LIN {X 0,Y 584.039,Z 358.291,A -85,B 0,C 180,E1 26452.128,E2 26452.128} C_VEL
LIN {X 0,Y 584.089,Z 358.294,A -85,B 0,C 180,E1 26449.046,E2 26449.046} C_VEL
LIN {X 0,Y 584.1,Z 358.289,A -85,B 0,C 180,E1 26446.664,E2 26446.664} C_VEL
LIN {X 0,Y 583.093,Z 358.412,A -85,B 0,C 180,E1 26445.909,E2 26445.909} C_VEL
LIN {X 0,Y 576.621,Z 359.216,A -85,B 0,C 180,E1 26443.789,E2 26443.789} C_VEL
LIN {X 0,Y 576.118,Z 359.28,A -85,B 0,C 180,E1 26443.236,E2 26443.236} C_VEL
LIN {X 0,Y 576.115,Z 359.276,A -85,B 0,C 180,E1 26439.857,E2 26439.857} C_VEL
LIN {X 0,Y 576.157,Z 359.281,A -85,B 0,C 180,E1 26436.692,E2 26436.692} C_VEL
LIN {X 0,Y 576.112,Z 359.278,A -85,B 0,C 180,E1 26433.51,E2 26433.51} C_VEL
LIN {X 0,Y 576.159,Z 359.278,A -85,B 0,C 180,E1 26430.357,E2 26430.357} C_VEL
LIN {X 0,Y 576.115,Z 359.28,A -85,B 0,C 180,E1 26427.131,E2 26427.131} C_VEL
LIN {X 0,Y 576.159,Z 359.276,A -85,B 0,C 180,E1 26423.961,E2 26423.961} C_VEL
LIN {X 0,Y 576.126,Z 359.281,A -85,B 0,C 180,E1 26420.71,E2 26420.71} C_VEL
LIN {X 0,Y 576.141,Z 359.275,A -85,B 0,C 180,E1 26417.371,E2 26417.371} C_VEL
LIN {X 0,Y 576.158,Z 359.281,A -85,B 0,C 180,E1 26414.073,E2 26414.073} C_VEL
LIN {X 0,Y 576.126,Z 359.278,A -85,B 0,C 180,E1 26410.828,E2 26410.828} C_VEL
LIN {X 0,Y 576.153,Z 359.277,A -85,B 0,C 180,E1 26407.647,E2 26407.647} C_VEL
LIN {X 0,Y 576.129,Z 359.278,A -85,B 0,C 180,E1 26404.451,E2 26404.451} C_VEL
LIN {X 0,Y 576.155,Z 359.268,A -85,B 0,C 180,E1 26401.179,E2 26401.179} C_VEL
LIN {X 0,Y 576.151,Z 359.283,A -85,B 0,C 180,E1 26397.824,E2 26397.824} C_VEL
LIN {X 0,Y 576.139,Z 359.274,A -85,B 0,C 180,E1 26394.501,E2 26394.501} C_VEL
LIN {X 0,Y 576.147,Z 359.275,A -85,B 0,C 180,E1 26391.263,E2 26391.263} C_VEL
LIN {X 0,Y 576.137,Z 359.279,A -85,B 0,C 180,E1 26388.005,E2 26388.005} C_VEL
LIN {X 0,Y 576.147,Z 359.274,A -85,B 0,C 180,E1 26384.777,E2 26384.777} C_VEL
LIN {X 0,Y 576.155,Z 359.274,A -85,B 0,C 180,E1 26381.407,E2 26381.407} C_VEL
LIN {X 0,Y 576.142,Z 359.208,A -85,B 0,C 180,E1 26378.078,E2 26378.078} C_VEL
LIN {X 0,Y 576.158,Z 359.375,A -85,B 0,C 180,E1 26377.927,E2 26377.927} C_VEL
LIN {X 0,Y 577.241,Z 362.387,A -85,B 0,C 180,E1 26377.662,E2 26377.662} C_VEL
LIN {X 0,Y 582.65,Z 371.03,A -85,B 0,C 180,E1 26377.087,E2 26377.087} C_VEL
LIN {X 0,Y 581.664,Z 577.888,A -85,B 0,C 180,E1 26374.006,E2 26374.006} C_VEL
LIN {X 0,Y 581.046,Z 710.787,A -85,B 0,C 180,E1 26372.053,E2 26372.053} C_VEL
LIN {X 0,Y 580.711,Z 734.473,A -85,B 0,C 180,E1 26371.508,E2 26371.508} C_VEL
LIN {X 0,Y 580.382,Z 757.042,A -85,B 0,C 180,E1 26370.799,E2 26370.799} C_VEL
LIN {X 0,Y 579.899,Z 779.356,A -85,B 0,C 180,E1 26369.899,E2 26369.899} C_VEL
LIN {X 0,Y 579.46,Z 801.416,A -85,B 0,C 180,E1 26368.811,E2 26368.811} C_VEL
LIN {X 0,Y 578.932,Z 822.341,A -85,B 0,C 180,E1 26367.572,E2 26367.572} C_VEL
LIN {X 0,Y 578.395,Z 843.774,A -85,B 0,C 180,E1 26366.082,E2 26366.082} C_VEL
LIN {X 0,Y 577.938,Z 863.519,A -85,B 0,C 180,E1 26364.488,E2 26364.488} C_VEL
LIN {X 0,Y 577.457,Z 882.263,A -85,B 0,C 180,E1 26362.736,E2 26362.736} C_VEL
LIN {X 0,Y 577.064,Z 899.119,A -85,B 0,C 180,E1 26360.926,E2 26360.926} C_VEL
LIN {X 0,Y 576.751,Z 914.853,A -85,B 0,C 180,E1 26359.004,E2 26359.004} C_VEL
LIN {X 0,Y 576.471,Z 928.62,A -85,B 0,C 180,E1 26357.069,E2 26357.069} C_VEL
LIN {X 0,Y 576.257,Z 941.929,A -85,B 0,C 180,E1 26354.912,E2 26354.912} C_VEL
LIN {X 0,Y 576.123,Z 952.394,A -85,B 0,C 180,E1 26352.942,E2 26352.942} C_VEL
LIN {X 0,Y 576.028,Z 962.321,A -85,B 0,C 180,E1 26350.741,E2 26350.741} C_VEL
LIN {X 0,Y 575.96,Z 970.279,A -85,B 0,C 180,E1 26348.618,E2 26348.618} C_VEL
LIN {X 0,Y 575.904,Z 977.029,A -85,B 0,C 180,E1 26346.354,E2 26346.354} C_VEL
LIN {X 0,Y 575.92,Z 981.572,A -85,B 0,C 180,E1 26344.385,E2 26344.385} C_VEL
LIN {X 0,Y 575.898,Z 985.394,A -85,B 0,C 180,E1 26342.044,E2 26342.044} C_VEL
LIN {X 0,Y 575.883,Z 987.298,A -85,B 0,C 180,E1 26339.996,E2 26339.996} C_VEL
LIN {X 0,Y 575.903,Z 987.961,A -85,B 0,C 180,E1 26337.727,E2 26337.727} C_VEL
LIN {X 0,Y 575.902,Z 987.038,A -85,B 0,C 180,E1 26335.527,E2 26335.527} C_VEL
LIN {X 0,Y 575.89,Z 984.436,A -85,B 0,C 180,E1 26333.167,E2 26333.167} C_VEL
LIN {X 0,Y 575.915,Z 980.609,A -85,B 0,C 180,E1 26331.058,E2 26331.058} C_VEL
LIN {X 0,Y 575.953,Z 974.751,A -85,B 0,C 180,E1 26328.723,E2 26328.723} C_VEL
LIN {X 0,Y 575.974,Z 968.076,A -85,B 0,C 180,E1 26326.666,E2 26326.666} C_VEL
LIN {X 0,Y 576.074,Z 958.832,A -85,B 0,C 180,E1 26324.348,E2 26324.348} C_VEL
LIN {X 0,Y 576.185,Z 948.859,A -85,B 0,C 180,E1 26322.269,E2 26322.269} C_VEL
LIN {X 0,Y 576.358,Z 936.393,A -85,B 0,C 180,E1 26320.062,E2 26320.062} C_VEL
LIN {X 0,Y 576.611,Z 922.852,A -85,B 0,C 180,E1 26317.994,E2 26317.994} C_VEL
LIN {X 0,Y 576.89,Z 907.932,A -85,B 0,C 180,E1 26316.031,E2 26316.031} C_VEL
LIN {X 0,Y 577.257,Z 890.405,A -85,B 0,C 180,E1 26314.019,E2 26314.019} C_VEL
LIN {X 0,Y 577.709,Z 872.006,A -85,B 0,C 180,E1 26312.184,E2 26312.184} C_VEL
LIN {X 0,Y 578.204,Z 852.474,A -85,B 0,C 180,E1 26310.5,E2 26310.5} C_VEL
LIN {X 0,Y 578.672,Z 832.219,A -85,B 0,C 180,E1 26308.996,E2 26308.996} C_VEL
LIN {X 0,Y 579.218,Z 811.476,A -85,B 0,C 180,E1 26307.669,E2 26307.669} C_VEL
LIN {X 0,Y 579.693,Z 789.853,A -85,B 0,C 180,E1 26306.503,E2 26306.503} C_VEL
LIN {X 0,Y 580.171,Z 767.04,A -85,B 0,C 180,E1 26305.492,E2 26305.492} C_VEL
LIN {X 0,Y 580.575,Z 744.527,A -85,B 0,C 180,E1 26304.692,E2 26304.692} C_VEL
LIN {X 0,Y 580.896,Z 721.993,A -85,B 0,C 180,E1 26304.092,E2 26304.092} C_VEL
LIN {X 0,Y 581.126,Z 699.044,A -85,B 0,C 180,E1 26303.661,E2 26303.661} C_VEL
LIN {X 0,Y 582.089,Z 486.06,A -85,B 0,C 180,E1 26300.55,E2 26300.55} C_VEL
LIN {X 0,Y 582.554,Z 370.789,A -85,B 0,C 180,E1 26298.812,E2 26298.812} C_VEL
LIN {X 0,Y 576.61,Z 361.104,A -85,B 0,C 180,E1 26298.147,E2 26298.147} C_VEL
LIN {X 0,Y 576.167,Z 359.389,A -85,B 0,C 180,E1 26297.918,E2 26297.918} C_VEL
LIN {X 0,Y 576.134,Z 359.254,A -85,B 0,C 180,E1 26294.678,E2 26294.678} C_VEL
LIN {X 0,Y 576.156,Z 359.272,A -85,B 0,C 180,E1 26291.309,E2 26291.309} C_VEL
LIN {X 0,Y 576.149,Z 359.282,A -85,B 0,C 180,E1 26287.981,E2 26287.981} C_VEL
LIN {X 0,Y 576.143,Z 359.279,A -85,B 0,C 180,E1 26284.679,E2 26284.679} C_VEL
LIN {X 0,Y 576.138,Z 359.278,A -85,B 0,C 180,E1 26281.492,E2 26281.492} C_VEL
LIN {X 0,Y 576.156,Z 359.283,A -85,B 0,C 180,E1 26278.21,E2 26278.21} C_VEL
LIN {X 0,Y 576.155,Z 359.272,A -85,B 0,C 180,E1 26274.823,E2 26274.823} C_VEL
LIN {X 0,Y 576.126,Z 359.28,A -85,B 0,C 180,E1 26271.517,E2 26271.517} C_VEL
LIN {X 0,Y 576.157,Z 359.279,A -85,B 0,C 180,E1 26268.286,E2 26268.286} C_VEL
LIN {X 0,Y 576.117,Z 359.279,A -85,B 0,C 180,E1 26265.117,E2 26265.117} C_VEL
LIN {X 0,Y 576.157,Z 359.283,A -85,B 0,C 180,E1 26261.903,E2 26261.903} C_VEL
LIN {X 0,Y 576.117,Z 359.279,A -85,B 0,C 180,E1 26258.733,E2 26258.733} C_VEL
LIN {X 0,Y 576.113,Z 359.283,A -85,B 0,C 180,E1 26255.385,E2 26255.385} C_VEL
LIN {X 0,Y 576.137,Z 359.279,A -85,B 0,C 180,E1 26252.263,E2 26252.263} C_VEL
LIN {X 0,Y 576.09,Z 359.283,A -85,B 0,C 180,E1 26249.026,E2 26249.026} C_VEL
LIN {X 0,Y 576.157,Z 359.282,A -85,B 0,C 180,E1 26245.873,E2 26245.873} C_VEL
LIN {X 0,Y 576.076,Z 359.284,A -85,B 0,C 180,E1 26242.719,E2 26242.719} C_VEL
LIN {X 0,Y 576.156,Z 359.281,A -85,B 0,C 180,E1 26239.628,E2 26239.628} C_VEL
LIN {X 0,Y 576.077,Z 359.287,A -85,B 0,C 180,E1 26236.446,E2 26236.446} C_VEL
LIN {X 0,Y 576.133,Z 359.273,A -85,B 0,C 180,E1 26233.277,E2 26233.277} C_VEL
LIN {X 0,Y 576.121,Z 359.484,A -85,B 0,C 180,E1 26232.179,E2 26232.179} C_VEL
LIN {X 0,Y 577.585,Z 362.94,A -85,B 0,C 180,E1 26231.746,E2 26231.746} C_VEL
LIN {X 0,Y 581.447,Z 371.701,A -85,B 0,C 180,E1 26230.768,E2 26230.768} C_VEL
LIN {X 0,Y 581.237,Z 391.484,A -85,B 0,C 180,E1 26229.398,E2 26229.398} C_VEL
LIN {X 0,Y 582.659,Z 399.132,A -85,B 0,C 180,E1 26229.161,E2 26229.161} C_VEL
LIN {X 0,Y 581.676,Z 605.241,A -85,B 0,C 180,E1 26226.09,E2 26226.09} C_VEL
LIN {X 0,Y 581.042,Z 739.782,A -85,B 0,C 180,E1 26224.112,E2 26224.112} C_VEL
LIN {X 0,Y 580.713,Z 763.541,A -85,B 0,C 180,E1 26223.576,E2 26223.576} C_VEL
LIN {X 0,Y 580.42,Z 784.658,A -85,B 0,C 180,E1 26222.925,E2 26222.925} C_VEL
LIN {X 0,Y 579.922,Z 807.644,A -85,B 0,C 180,E1 26222.019,E2 26222.019} C_VEL
LIN {X 0,Y 579.517,Z 829.396,A -85,B 0,C 180,E1 26220.965,E2 26220.965} C_VEL
LIN {X 0,Y 578.968,Z 849.901,A -85,B 0,C 180,E1 26219.771,E2 26219.771} C_VEL
LIN {X 0,Y 578.481,Z 871.122,A -85,B 0,C 180,E1 26218.325,E2 26218.325} C_VEL
LIN {X 0,Y 577.996,Z 889.886,A -85,B 0,C 180,E1 26216.842,E2 26216.842} C_VEL
LIN {X 0,Y 577.557,Z 907.885,A -85,B 0,C 180,E1 26215.208,E2 26215.208} C_VEL
LIN {X 0,Y 577.192,Z 924.958,A -85,B 0,C 180,E1 26213.448,E2 26213.448} C_VEL
LIN {X 0,Y 576.817,Z 940.828,A -85,B 0,C 180,E1 26211.562,E2 26211.562} C_VEL
LIN {X 0,Y 576.519,Z 956.319,A -85,B 0,C 180,E1 26209.452,E2 26209.452} C_VEL
LIN {X 0,Y 576.323,Z 969.345,A -85,B 0,C 180,E1 26207.411,E2 26207.411} C_VEL
LIN {X 0,Y 576.149,Z 980.826,A -85,B 0,C 180,E1 26205.297,E2 26205.297} C_VEL
LIN {X 0,Y 576.036,Z 990.871,A -85,B 0,C 180,E1 26203.145,E2 26203.145} C_VEL
LIN {X 0,Y 575.953,Z 999.043,A -85,B 0,C 180,E1 26201.011,E2 26201.011} C_VEL
LIN {X 0,Y 575.942,Z 1005.768,A -85,B 0,C 180,E1 26198.891,E2 26198.891} C_VEL
LIN {X 0,Y 575.907,Z 1011.042,A -85,B 0,C 180,E1 26196.682,E2 26196.682} C_VEL
LIN {X 0,Y 575.902,Z 1014.909,A -85,B 0,C 180,E1 26194.483,E2 26194.483} C_VEL
LIN {X 0,Y 575.915,Z 1017.187,A -85,B 0,C 180,E1 26192.191,E2 26192.191} C_VEL
LIN {X 0,Y 575.908,Z 1018,A -85,B 0,C 180,E1 26190.003,E2 26190.003} C_VEL
LIN {X 0,Y 575.915,Z 1017.191,A -85,B 0,C 180,E1 26187.814,E2 26187.814} C_VEL
LIN {X 0,Y 575.901,Z 1014.917,A -85,B 0,C 180,E1 26185.522,E2 26185.522} C_VEL
LIN {X 0,Y 575.908,Z 1011.053,A -85,B 0,C 180,E1 26183.323,E2 26183.323} C_VEL
LIN {X 0,Y 575.944,Z 1005.561,A -85,B 0,C 180,E1 26181.039,E2 26181.039} C_VEL
LIN {X 0,Y 575.956,Z 998.705,A -85,B 0,C 180,E1 26178.893,E2 26178.893} C_VEL
LIN {X 0,Y 576.039,Z 990.47,A -85,B 0,C 180,E1 26176.758,E2 26176.758} C_VEL
LIN {X 0,Y 576.15,Z 980.854,A -85,B 0,C 180,E1 26174.709,E2 26174.709} C_VEL
LIN {X 0,Y 576.323,Z 969.347,A -85,B 0,C 180,E1 26172.589,E2 26172.589} C_VEL
LIN {X 0,Y 576.518,Z 956.356,A -85,B 0,C 180,E1 26170.553,E2 26170.553} C_VEL
LIN {X 0,Y 576.814,Z 940.872,A -85,B 0,C 180,E1 26168.443,E2 26168.443} C_VEL
LIN {X 0,Y 577.197,Z 924.708,A -85,B 0,C 180,E1 26166.524,E2 26166.524} C_VEL
LIN {X 0,Y 577.573,Z 907.39,A -85,B 0,C 180,E1 26164.744,E2 26164.744} C_VEL
LIN {X 0,Y 578.038,Z 887.68,A -85,B 0,C 180,E1 26162.975,E2 26162.975} C_VEL
LIN {X 0,Y 578.573,Z 868.244,A -85,B 0,C 180,E1 26161.46,E2 26161.46} C_VEL
LIN {X 0,Y 579.038,Z 847.694,A -85,B 0,C 180,E1 26160.092,E2 26160.092} C_VEL
LIN {X 0,Y 579.566,Z 825.51,A -85,B 0,C 180,E1 26158.836,E2 26158.836} C_VEL
LIN {X 0,Y 579.994,Z 805.223,A -85,B 0,C 180,E1 26157.875,E2 26157.875} C_VEL
LIN {X 0,Y 580.438,Z 782.309,A -85,B 0,C 180,E1 26156.995,E2 26156.995} C_VEL
LIN {X 0,Y 580.746,Z 761.445,A -85,B 0,C 180,E1 26156.366,E2 26156.366} C_VEL
LIN {X 0,Y 581.048,Z 738.298,A -85,B 0,C 180,E1 26155.862,E2 26155.862} C_VEL
LIN {X 0,Y 582.086,Z 514.845,A -85,B 0,C 180,E1 26152.576,E2 26152.576} C_VEL
LIN {X 0,Y 582.507,Z 397.408,A -85,B 0,C 180,E1 26150.8,E2 26150.8} C_VEL
LIN {X 0,Y 581.157,Z 390.899,A -85,B 0,C 180,E1 26150.577,E2 26150.577} C_VEL
LIN {X 0,Y 581.328,Z 371.136,A -85,B 0,C 180,E1 26149.181,E2 26149.181} C_VEL
LIN {X 0,Y 577.109,Z 362.215,A -85,B 0,C 180,E1 26148.157,E2 26148.157} C_VEL
LIN {X 0,Y 576.109,Z 359.405,A -85,B 0,C 180,E1 26147.79,E2 26147.79} C_VEL
LIN {X 0,Y 576.104,Z 359.273,A -85,B 0,C 180,E1 26144.925,E2 26144.925} C_VEL
LIN {X 0,Y 576.087,Z 359.286,A -85,B 0,C 180,E1 26141.585,E2 26141.585} C_VEL
LIN {X 0,Y 576.109,Z 359.275,A -85,B 0,C 180,E1 26138.655,E2 26138.655} C_VEL
LIN {X 0,Y 576.082,Z 359.273,A -85,B 0,C 180,E1 26135.429,E2 26135.429} C_VEL
LIN {X 0,Y 576.102,Z 359.284,A -85,B 0,C 180,E1 26132.499,E2 26132.499} C_VEL
LIN {X 0,Y 576.079,Z 359.281,A -85,B 0,C 180,E1 26129.304,E2 26129.304} C_VEL
LIN {X 0,Y 576.083,Z 359.284,A -85,B 0,C 180,E1 26126.49,E2 26126.49} C_VEL
LIN {X 0,Y 576.08,Z 359.282,A -85,B 0,C 180,E1 26123.094,E2 26123.094} C_VEL
LIN {X 0,Y 576.098,Z 359.283,A -85,B 0,C 180,E1 26120.205,E2 26120.205} C_VEL
LIN {X 0,Y 576.088,Z 359.282,A -85,B 0,C 180,E1 26116.952,E2 26116.952} C_VEL
LIN {X 0,Y 576.1,Z 359.282,A -85,B 0,C 180,E1 26114.047,E2 26114.047} C_VEL
LIN {X 0,Y 576.088,Z 359.281,A -85,B 0,C 180,E1 26110.702,E2 26110.702} C_VEL
LIN {X 0,Y 576.126,Z 359.283,A -85,B 0,C 180,E1 26107.679,E2 26107.679} C_VEL
LIN {X 0,Y 576.092,Z 359.279,A -85,B 0,C 180,E1 26104.479,E2 26104.479} C_VEL
LIN {X 0,Y 576.145,Z 359.283,A -85,B 0,C 180,E1 26101.392,E2 26101.392} C_VEL
LIN {X 0,Y 576.094,Z 359.28,A -85,B 0,C 180,E1 26098.209,E2 26098.209} C_VEL
LIN {X 0,Y 576.157,Z 359.281,A -85,B 0,C 180,E1 26095.122,E2 26095.122} C_VEL
LIN {X 0,Y 576.097,Z 359.281,A -85,B 0,C 180,E1 26091.918,E2 26091.918} C_VEL
LIN {X 0,Y 576.162,Z 359.278,A -85,B 0,C 180,E1 26088.691,E2 26088.691} C_VEL
LIN {X 0,Y 576.106,Z 359.281,A -85,B 0,C 180,E1 26085.527,E2 26085.527} C_VEL
LIN {X 0,Y 576.118,Z 359.28,A -85,B 0,C 180,E1 26083.236,E2 26083.236} C_VEL
LIN {X 0,Y 575.172,Z 359.405,A -85,B 0,C 180,E1 26082.47,E2 26082.47} C_VEL
LIN {X 0,Y 568.624,Z 360.213,A -85,B 0,C 180,E1 26080.264,E2 26080.264} C_VEL
LIN {X 0,Y 568.172,Z 360.265,A -85,B 0,C 180,E1 26079.76,E2 26079.76} C_VEL
LIN {X 0,Y 568.223,Z 360.268,A -85,B 0,C 180,E1 26076.567,E2 26076.567} C_VEL
LIN {X 0,Y 568.172,Z 360.268,A -85,B 0,C 180,E1 26073.337,E2 26073.337} C_VEL
LIN {X 0,Y 568.222,Z 360.263,A -85,B 0,C 180,E1 26070.134,E2 26070.134} C_VEL
LIN {X 0,Y 568.184,Z 360.27,A -85,B 0,C 180,E1 26066.883,E2 26066.883} C_VEL
LIN {X 0,Y 568.195,Z 360.265,A -85,B 0,C 180,E1 26063.503,E2 26063.503} C_VEL
LIN {X 0,Y 568.219,Z 360.27,A -85,B 0,C 180,E1 26060.254,E2 26060.254} C_VEL
LIN {X 0,Y 568.183,Z 360.267,A -85,B 0,C 180,E1 26056.938,E2 26056.938} C_VEL
LIN {X 0,Y 568.218,Z 360.263,A -85,B 0,C 180,E1 26053.679,E2 26053.679} C_VEL
LIN {X 0,Y 568.197,Z 360.27,A -85,B 0,C 180,E1 26050.354,E2 26050.354} C_VEL
LIN {X 0,Y 568.201,Z 360.263,A -85,B 0,C 180,E1 26046.974,E2 26046.974} C_VEL
LIN {X 0,Y 568.215,Z 360.27,A -85,B 0,C 180,E1 26043.657,E2 26043.657} C_VEL
LIN {X 0,Y 568.191,Z 360.26,A -85,B 0,C 180,E1 26040.428,E2 26040.428} C_VEL
LIN {X 0,Y 568.212,Z 360.263,A -85,B 0,C 180,E1 26037.223,E2 26037.223} C_VEL
LIN {X 0,Y 568.2,Z 360.267,A -85,B 0,C 180,E1 26033.981,E2 26033.981} C_VEL
LIN {X 0,Y 568.216,Z 360.26,A -85,B 0,C 180,E1 26030.588,E2 26030.588} C_VEL
LIN {X 0,Y 568.212,Z 360.262,A -85,B 0,C 180,E1 26027.297,E2 26027.297} C_VEL
LIN {X 0,Y 568.202,Z 360.26,A -85,B 0,C 180,E1 26024.051,E2 26024.051} C_VEL
LIN {X 0,Y 568.206,Z 360.27,A -85,B 0,C 180,E1 26020.747,E2 26020.747} C_VEL
LIN {X 0,Y 568.237,Z 360.461,A -85,B 0,C 180,E1 26018.549,E2 26018.549} C_VEL
LIN {X 0,Y 568.612,Z 361.903,A -85,B 0,C 180,E1 26018.396,E2 26018.396} C_VEL
LIN {X 0,Y 570.597,Z 364.971,A -85,B 0,C 180,E1 26018.176,E2 26018.176} C_VEL
LIN {X 0,Y 576.417,Z 374.479,A -85,B 0,C 180,E1 26017.538,E2 26017.538} C_VEL
LIN {X 0,Y 575.172,Z 581.534,A -85,B 0,C 180,E1 26014.423,E2 26014.423} C_VEL
LIN {X 0,Y 574.41,Z 710.851,A -85,B 0,C 180,E1 26012.501,E2 26012.501} C_VEL
LIN {X 0,Y 573.992,Z 734.738,A -85,B 0,C 180,E1 26011.947,E2 26011.947} C_VEL
LIN {X 0,Y 573.561,Z 757.89,A -85,B 0,C 180,E1 26011.208,E2 26011.208} C_VEL
LIN {X 0,Y 572.966,Z 780.111,A -85,B 0,C 180,E1 26010.297,E2 26010.297} C_VEL
LIN {X 0,Y 572.368,Z 802.944,A -85,B 0,C 180,E1 26009.147,E2 26009.147} C_VEL
LIN {X 0,Y 571.724,Z 823.729,A -85,B 0,C 180,E1 26007.893,E2 26007.893} C_VEL
LIN {X 0,Y 571.079,Z 844.306,A -85,B 0,C 180,E1 26006.434,E2 26006.434} C_VEL
LIN {X 0,Y 570.482,Z 864.001,A -85,B 0,C 180,E1 26004.819,E2 26004.819} C_VEL
LIN {X 0,Y 569.873,Z 882.699,A -85,B 0,C 180,E1 26003.044,E2 26003.044} C_VEL
LIN {X 0,Y 569.387,Z 899.492,A -85,B 0,C 180,E1 26001.21,E2 26001.21} C_VEL
LIN {X 0,Y 568.971,Z 915.513,A -85,B 0,C 180,E1 25999.216,E2 25999.216} C_VEL
LIN {X 0,Y 568.614,Z 930.281,A -85,B 0,C 180,E1 25997.094,E2 25997.094} C_VEL
LIN {X 0,Y 568.345,Z 942.905,A -85,B 0,C 180,E1 25994.979,E2 25994.979} C_VEL
LIN {X 0,Y 568.172,Z 953.893,A -85,B 0,C 180,E1 25992.856,E2 25992.856} C_VEL
LIN {X 0,Y 568.041,Z 963.441,A -85,B 0,C 180,E1 25990.642,E2 25990.642} C_VEL
LIN {X 0,Y 567.982,Z 971.665,A -85,B 0,C 180,E1 25988.354,E2 25988.354} C_VEL
LIN {X 0,Y 567.91,Z 977.661,A -85,B 0,C 180,E1 25986.221,E2 25986.221} C_VEL
LIN {X 0,Y 567.901,Z 982.322,A -85,B 0,C 180,E1 25984.109,E2 25984.109} C_VEL
LIN {X 0,Y 567.911,Z 985.811,A -85,B 0,C 180,E1 25981.73,E2 25981.73} C_VEL
LIN {X 0,Y 567.892,Z 987.616,A -85,B 0,C 180,E1 25979.53,E2 25979.53} C_VEL
LIN {X 0,Y 567.896,Z 987.864,A -85,B 0,C 180,E1 25977.279,E2 25977.279} C_VEL
LIN {X 0,Y 567.915,Z 986.645,A -85,B 0,C 180,E1 25974.952,E2 25974.952} C_VEL
LIN {X 0,Y 567.912,Z 983.846,A -85,B 0,C 180,E1 25972.723,E2 25972.723} C_VEL
LIN {X 0,Y 567.937,Z 979.456,A -85,B 0,C 180,E1 25970.407,E2 25970.407} C_VEL
LIN {X 0,Y 567.951,Z 973.383,A -85,B 0,C 180,E1 25968.132,E2 25968.132} C_VEL
LIN {X 0,Y 568.016,Z 965.575,A -85,B 0,C 180,E1 25965.806,E2 25965.806} C_VEL
LIN {X 0,Y 568.135,Z 956.454,A -85,B 0,C 180,E1 25963.621,E2 25963.621} C_VEL
LIN {X 0,Y 568.321,Z 944.838,A -85,B 0,C 180,E1 25961.281,E2 25961.281} C_VEL
LIN {X 0,Y 568.588,Z 932.385,A -85,B 0,C 180,E1 25959.146,E2 25959.146} C_VEL
LIN {X 0,Y 568.91,Z 917.928,A -85,B 0,C 180,E1 25957.026,E2 25957.026} C_VEL
LIN {X 0,Y 569.311,Z 902.501,A -85,B 0,C 180,E1 25955.051,E2 25955.051} C_VEL
LIN {X 0,Y 569.816,Z 885.708,A -85,B 0,C 180,E1 25953.174,E2 25953.174} C_VEL
LIN {X 0,Y 570.37,Z 867.196,A -85,B 0,C 180,E1 25951.381,E2 25951.381} C_VEL
LIN {X 0,Y 570.972,Z 847.303,A -85,B 0,C 180,E1 25949.705,E2 25949.705} C_VEL
LIN {X 0,Y 571.646,Z 827.089,A -85,B 0,C 180,E1 25948.238,E2 25948.238} C_VEL
LIN {X 0,Y 572.247,Z 806.14,A -85,B 0,C 180,E1 25946.944,E2 25946.944} C_VEL
LIN {X 0,Y 572.897,Z 784.492,A -85,B 0,C 180,E1 25945.814,E2 25945.814} C_VEL
LIN {X 0,Y 573.405,Z 762.546,A -85,B 0,C 180,E1 25944.877,E2 25944.877} C_VEL
LIN {X 0,Y 573.946,Z 739.05,A -85,B 0,C 180,E1 25944.085,E2 25944.085} C_VEL
LIN {X 0,Y 574.303,Z 716.026,A -85,B 0,C 180,E1 25943.51,E2 25943.51} C_VEL
LIN {X 0,Y 574.59,Z 685.111,A -85,B 0,C 180,E1 25943.006,E2 25943.006} C_VEL
LIN {X 0,Y 575.802,Z 474.249,A -85,B 0,C 180,E1 25939.887,E2 25939.887} C_VEL
LIN {X 0,Y 576.295,Z 374.09,A -85,B 0,C 180,E1 25938.356,E2 25938.356} C_VEL
LIN {X 0,Y 570.238,Z 364.653,A -85,B 0,C 180,E1 25937.698,E2 25937.698} C_VEL
LIN {X 0,Y 568.425,Z 361.357,A -85,B 0,C 180,E1 25937.479,E2 25937.479} C_VEL
LIN {X 0,Y 568.212,Z 360.355,A -85,B 0,C 180,E1 25937.301,E2 25937.301} C_VEL
LIN {X 0,Y 568.211,Z 360.245,A -85,B 0,C 180,E1 25934.054,E2 25934.054} C_VEL
LIN {X 0,Y 568.197,Z 360.262,A -85,B 0,C 180,E1 25930.853,E2 25930.853} C_VEL
LIN {X 0,Y 568.207,Z 360.267,A -85,B 0,C 180,E1 25927.584,E2 25927.584} C_VEL
LIN {X 0,Y 568.216,Z 360.27,A -85,B 0,C 180,E1 25924.239,E2 25924.239} C_VEL
LIN {X 0,Y 568.216,Z 360.265,A -85,B 0,C 180,E1 25920.908,E2 25920.908} C_VEL
LIN {X 0,Y 568.194,Z 360.268,A -85,B 0,C 180,E1 25917.58,E2 25917.58} C_VEL
LIN {X 0,Y 568.218,Z 360.268,A -85,B 0,C 180,E1 25914.244,E2 25914.244} C_VEL
LIN {X 0,Y 568.198,Z 360.266,A -85,B 0,C 180,E1 25910.99,E2 25910.99} C_VEL
LIN {X 0,Y 568.19,Z 360.271,A -85,B 0,C 180,E1 25907.596,E2 25907.596} C_VEL
LIN {X 0,Y 568.22,Z 360.266,A -85,B 0,C 180,E1 25904.382,E2 25904.382} C_VEL
LIN {X 0,Y 568.171,Z 360.269,A -85,B 0,C 180,E1 25901.107,E2 25901.107} C_VEL
LIN {X 0,Y 568.221,Z 360.271,A -85,B 0,C 180,E1 25897.88,E2 25897.88} C_VEL
LIN {X 0,Y 568.169,Z 360.27,A -85,B 0,C 180,E1 25894.683,E2 25894.683} C_VEL
LIN {X 0,Y 568.167,Z 360.27,A -85,B 0,C 180,E1 25891.287,E2 25891.287} C_VEL
LIN {X 0,Y 568.17,Z 360.271,A -85,B 0,C 180,E1 25888.371,E2 25888.371} C_VEL
LIN {X 0,Y 568.151,Z 360.274,A -85,B 0,C 180,E1 25885.095,E2 25885.095} C_VEL
LIN {X 0,Y 568.177,Z 360.273,A -85,B 0,C 180,E1 25882.036,E2 25882.036} C_VEL
LIN {X 0,Y 568.136,Z 360.276,A -85,B 0,C 180,E1 25878.838,E2 25878.838} C_VEL
LIN {X 0,Y 568.205,Z 360.265,A -85,B 0,C 180,E1 25875.686,E2 25875.686} C_VEL
LIN {X 0,Y 568.183,Z 360.486,A -85,B 0,C 180,E1 25872.832,E2 25872.832} C_VEL
LIN {X 0,Y 569.669,Z 364.048,A -85,B 0,C 180,E1 25872.377,E2 25872.377} C_VEL
LIN {X 0,Y 574.864,Z 375.383,A -85,B 0,C 180,E1 25871.064,E2 25871.064} C_VEL
LIN {X 0,Y 574.653,Z 391.507,A -85,B 0,C 180,E1 25869.939,E2 25869.939} C_VEL
LIN {X 0,Y 576.441,Z 400.852,A -85,B 0,C 180,E1 25869.639,E2 25869.639} C_VEL
LIN {X 0,Y 575.196,Z 607.171,A -85,B 0,C 180,E1 25866.533,E2 25866.533} C_VEL
LIN {X 0,Y 574.407,Z 739.89,A -85,B 0,C 180,E1 25864.56,E2 25864.56} C_VEL
LIN {X 0,Y 573.995,Z 763.697,A -85,B 0,C 180,E1 25864.018,E2 25864.018} C_VEL
LIN {X 0,Y 573.618,Z 785.253,A -85,B 0,C 180,E1 25863.346,E2 25863.346} C_VEL
LIN {X 0,Y 573.023,Z 807.646,A -85,B 0,C 180,E1 25862.451,E2 25862.451} C_VEL
LIN {X 0,Y 572.505,Z 828.753,A -85,B 0,C 180,E1 25861.423,E2 25861.423} C_VEL
LIN {X 0,Y 571.827,Z 849.905,A -85,B 0,C 180,E1 25860.181,E2 25860.181} C_VEL
LIN {X 0,Y 571.197,Z 871.113,A -85,B 0,C 180,E1 25858.721,E2 25858.721} C_VEL
LIN {X 0,Y 570.578,Z 889.888,A -85,B 0,C 180,E1 25857.219,E2 25857.219} C_VEL
LIN {X 0,Y 570.013,Z 908.438,A -85,B 0,C 180,E1 25855.51,E2 25855.51} C_VEL
LIN {X 0,Y 569.526,Z 925.6,A -85,B 0,C 180,E1 25853.707,E2 25853.707} C_VEL
LIN {X 0,Y 569.061,Z 941.677,A -85,B 0,C 180,E1 25851.763,E2 25851.763} C_VEL
LIN {X 0,Y 568.708,Z 956.32,A -85,B 0,C 180,E1 25849.73,E2 25849.73} C_VEL
LIN {X 0,Y 568.445,Z 968.996,A -85,B 0,C 180,E1 25847.718,E2 25847.718} C_VEL
LIN {X 0,Y 568.221,Z 980.307,A -85,B 0,C 180,E1 25845.62,E2 25845.62} C_VEL
LIN {X 0,Y 568.079,Z 989.987,A -85,B 0,C 180,E1 25843.54,E2 25843.54} C_VEL
LIN {X 0,Y 567.985,Z 998.483,A -85,B 0,C 180,E1 25841.329,E2 25841.329} C_VEL
LIN {X 0,Y 567.948,Z 1005.165,A -85,B 0,C 180,E1 25839.221,E2 25839.221} C_VEL
LIN {X 0,Y 567.895,Z 1010.629,A -85,B 0,C 180,E1 25836.98,E2 25836.98} C_VEL
LIN {X 0,Y 567.907,Z 1014.272,A -85,B 0,C 180,E1 25834.952,E2 25834.952} C_VEL
LIN {X 0,Y 567.915,Z 1016.986,A -85,B 0,C 180,E1 25832.525,E2 25832.525} C_VEL
LIN {X 0,Y 567.887,Z 1017.916,A -85,B 0,C 180,E1 25830.406,E2 25830.406} C_VEL
LIN {X 0,Y 567.913,Z 1017.325,A -85,B 0,C 180,E1 25827.985,E2 25827.985} C_VEL
LIN {X 0,Y 567.911,Z 1015.28,A -85,B 0,C 180,E1 25825.762,E2 25825.762} C_VEL
LIN {X 0,Y 567.918,Z 1011.466,A -85,B 0,C 180,E1 25823.432,E2 25823.432} C_VEL
LIN {X 0,Y 567.94,Z 1006.558,A -85,B 0,C 180,E1 25821.295,E2 25821.295} C_VEL
LIN {X 0,Y 567.969,Z 999.774,A -85,B 0,C 180,E1 25819.043,E2 25819.043} C_VEL
LIN {X 0,Y 568.067,Z 992.121,A -85,B 0,C 180,E1 25816.983,E2 25816.983} C_VEL
LIN {X 0,Y 568.211,Z 981.612,A -85,B 0,C 180,E1 25814.642,E2 25814.642} C_VEL
LIN {X 0,Y 568.423,Z 970.256,A -85,B 0,C 180,E1 25812.498,E2 25812.498} C_VEL
LIN {X 0,Y 568.669,Z 957.594,A -85,B 0,C 180,E1 25810.46,E2 25810.46} C_VEL
LIN {X 0,Y 569.03,Z 943.412,A -85,B 0,C 180,E1 25808.458,E2 25808.458} C_VEL
LIN {X 0,Y 569.448,Z 927.934,A -85,B 0,C 180,E1 25806.565,E2 25806.565} C_VEL
LIN {X 0,Y 569.948,Z 910.155,A -85,B 0,C 180,E1 25804.66,E2 25804.66} C_VEL
LIN {X 0,Y 570.534,Z 891.94,A -85,B 0,C 180,E1 25802.954,E2 25802.954} C_VEL
LIN {X 0,Y 571.139,Z 872.663,A -85,B 0,C 180,E1 25801.397,E2 25801.397} C_VEL
LIN {X 0,Y 571.758,Z 852.034,A -85,B 0,C 180,E1 25799.954,E2 25799.954} C_VEL
LIN {X 0,Y 572.398,Z 831.906,A -85,B 0,C 180,E1 25798.753,E2 25798.753} C_VEL
LIN {X 0,Y 572.972,Z 809.417,A -85,B 0,C 180,E1 25797.628,E2 25797.628} C_VEL
LIN {X 0,Y 573.579,Z 787.479,A -85,B 0,C 180,E1 25796.732,E2 25796.732} C_VEL
LIN {X 0,Y 573.979,Z 765.033,A -85,B 0,C 180,E1 25796.019,E2 25796.019} C_VEL
LIN {X 0,Y 574.39,Z 742.283,A -85,B 0,C 180,E1 25795.481,E2 25795.481} C_VEL
LIN {X 0,Y 574.733,Z 689.884,A -85,B 0,C 180,E1 25794.684,E2 25794.684} C_VEL
LIN {X 0,Y 575.912,Z 483.419,A -85,B 0,C 180,E1 25791.616,E2 25791.616} C_VEL
LIN {X 0,Y 576.28,Z 399.124,A -85,B 0,C 180,E1 25790.321,E2 25790.321} C_VEL
LIN {X 0,Y 574.55,Z 390.626,A -85,B 0,C 180,E1 25790.019,E2 25790.019} C_VEL
LIN {X 0,Y 574.864,Z 375.383,A -85,B 0,C 180,E1 25788.936,E2 25788.936} C_VEL
LIN {X 0,Y 569.72,Z 364.119,A -85,B 0,C 180,E1 25787.633,E2 25787.633} C_VEL
LIN {X 0,Y 568.194,Z 360.55,A -85,B 0,C 180,E1 25787.177,E2 25787.177} C_VEL
LIN {X 0,Y 568.177,Z 360.277,A -85,B 0,C 180,E1 25786.033,E2 25786.033} C_VEL
LIN {X 0,Y 568.15,Z 360.26,A -85,B 0,C 180,E1 25783.064,E2 25783.064} C_VEL
LIN {X 0,Y 568.156,Z 360.263,A -85,B 0,C 180,E1 25779.703,E2 25779.703} C_VEL
LIN {X 0,Y 568.156,Z 360.274,A -85,B 0,C 180,E1 25776.751,E2 25776.751} C_VEL
LIN {X 0,Y 568.145,Z 360.274,A -85,B 0,C 180,E1 25773.424,E2 25773.424} C_VEL
LIN {X 0,Y 568.159,Z 360.266,A -85,B 0,C 180,E1 25770.452,E2 25770.452} C_VEL
LIN {X 0,Y 568.139,Z 360.274,A -85,B 0,C 180,E1 25767.23,E2 25767.23} C_VEL
LIN {X 0,Y 568.158,Z 360.274,A -85,B 0,C 180,E1 25764.285,E2 25764.285} C_VEL
LIN {X 0,Y 568.143,Z 360.272,A -85,B 0,C 180,E1 25761.039,E2 25761.039} C_VEL
LIN {X 0,Y 568.171,Z 360.273,A -85,B 0,C 180,E1 25758.042,E2 25758.042} C_VEL
LIN {X 0,Y 568.145,Z 360.27,A -85,B 0,C 180,E1 25754.784,E2 25754.784} C_VEL
LIN {X 0,Y 568.185,Z 360.273,A -85,B 0,C 180,E1 25751.778,E2 25751.778} C_VEL
LIN {X 0,Y 568.147,Z 360.27,A -85,B 0,C 180,E1 25748.522,E2 25748.522} C_VEL
LIN {X 0,Y 568.21,Z 360.272,A -85,B 0,C 180,E1 25745.452,E2 25745.452} C_VEL
LIN {X 0,Y 568.151,Z 360.27,A -85,B 0,C 180,E1 25742.219,E2 25742.219} C_VEL
LIN {X 0,Y 568.222,Z 360.269,A -85,B 0,C 180,E1 25739.092,E2 25739.092} C_VEL
LIN {X 0,Y 568.156,Z 360.27,A -85,B 0,C 180,E1 25735.963,E2 25735.963} C_VEL
LIN {X 0,Y 568.215,Z 360.267,A -85,B 0,C 180,E1 25732.721,E2 25732.721} C_VEL
LIN {X 0,Y 568.166,Z 360.27,A -85,B 0,C 180,E1 25729.557,E2 25729.557} C_VEL
LIN {X 0,Y 568.186,Z 360.267,A -85,B 0,C 180,E1 25726.238,E2 25726.238} C_VEL
LIN {X 0,Y 568.19,Z 360.27,A -85,B 0,C 180,E1 25723.12,E2 25723.12} C_VEL
LIN {X 0,Y 568.174,Z 360.265,A -85,B 0,C 180,E1 25719.823,E2 25719.823} C_VEL
LIN {X 0,Y 568.172,Z 360.265,A -85,B 0,C 180,E1 25719.76,E2 25719.76} C_VEL
LIN {X 0,Y 567.184,Z 360.396,A -85,B 0,C 180,E1 25718.983,E2 25718.983} C_VEL
LIN {X 0,Y 560.731,Z 361.202,A -85,B 0,C 180,E1 25716.746,E2 25716.746} C_VEL
LIN {X 0,Y 560.28,Z 361.253,A -85,B 0,C 180,E1 25716.235,E2 25716.235} C_VEL
LIN {X 0,Y 560.241,Z 361.258,A -85,B 0,C 180,E1 25713.043,E2 25713.043} C_VEL
LIN {X 0,Y 560.251,Z 361.252,A -85,B 0,C 180,E1 25709.664,E2 25709.664} C_VEL
LIN {X 0,Y 560.279,Z 361.258,A -85,B 0,C 180,E1 25706.412,E2 25706.412} C_VEL
LIN {X 0,Y 560.238,Z 361.257,A -85,B 0,C 180,E1 25703.08,E2 25703.08} C_VEL
LIN {X 0,Y 560.283,Z 361.25,A -85,B 0,C 180,E1 25699.758,E2 25699.758} C_VEL
LIN {X 0,Y 560.263,Z 361.26,A -85,B 0,C 180,E1 25696.426,E2 25696.426} C_VEL
LIN {X 0,Y 560.256,Z 361.251,A -85,B 0,C 180,E1 25693.114,E2 25693.114} C_VEL
LIN {X 0,Y 560.279,Z 361.258,A -85,B 0,C 180,E1 25689.836,E2 25689.836} C_VEL
LIN {X 0,Y 560.25,Z 361.255,A -85,B 0,C 180,E1 25686.573,E2 25686.573} C_VEL
LIN {X 0,Y 560.279,Z 361.253,A -85,B 0,C 180,E1 25683.216,E2 25683.216} C_VEL
LIN {X 0,Y 560.276,Z 361.249,A -85,B 0,C 180,E1 25679.852,E2 25679.852} C_VEL
LIN {X 0,Y 560.259,Z 361.252,A -85,B 0,C 180,E1 25676.493,E2 25676.493} C_VEL
LIN {X 0,Y 560.27,Z 361.256,A -85,B 0,C 180,E1 25673.209,E2 25673.209} C_VEL
LIN {X 0,Y 560.265,Z 361.255,A -85,B 0,C 180,E1 25669.865,E2 25669.865} C_VEL
LIN {X 0,Y 560.279,Z 361.251,A -85,B 0,C 180,E1 25666.481,E2 25666.481} C_VEL
LIN {X 0,Y 560.266,Z 361.229,A -85,B 0,C 180,E1 25663.096,E2 25663.096} C_VEL
LIN {X 0,Y 560.261,Z 361.239,A -85,B 0,C 180,E1 25659.862,E2 25659.862} C_VEL
LIN {X 0,Y 560.305,Z 361.455,A -85,B 0,C 180,E1 25659.239,E2 25659.239} C_VEL
LIN {X 0,Y 560.637,Z 362.812,A -85,B 0,C 180,E1 25659.079,E2 25659.079} C_VEL
LIN {X 0,Y 562.509,Z 365.834,A -85,B 0,C 180,E1 25658.862,E2 25658.862} C_VEL
LIN {X 0,Y 563.758,Z 367.57,A -85,B 0,C 180,E1 25658.724,E2 25658.724} C_VEL
LIN {X 0,Y 570.223,Z 377.822,A -85,B 0,C 180,E1 25658.001,E2 25658.001} C_VEL
LIN {X 0,Y 568.709,Z 585.599,A -85,B 0,C 180,E1 25654.843,E2 25654.843} C_VEL
LIN {X 0,Y 567.81,Z 710.911,A -85,B 0,C 180,E1 25652.959,E2 25652.959} C_VEL
LIN {X 0,Y 567.314,Z 734.774,A -85,B 0,C 180,E1 25652.403,E2 25652.403} C_VEL
LIN {X 0,Y 566.785,Z 758.215,A -85,B 0,C 180,E1 25651.646,E2 25651.646} C_VEL
LIN {X 0,Y 566.097,Z 779.747,A -85,B 0,C 180,E1 25650.756,E2 25650.756} C_VEL
LIN {X 0,Y 565.408,Z 801.814,A -85,B 0,C 180,E1 25649.643,E2 25649.643} C_VEL
LIN {X 0,Y 564.603,Z 822.772,A -85,B 0,C 180,E1 25648.374,E2 25648.374} C_VEL
LIN {X 0,Y 563.843,Z 843.517,A -85,B 0,C 180,E1 25646.897,E2 25646.897} C_VEL
LIN {X 0,Y 563.076,Z 863.334,A -85,B 0,C 180,E1 25645.261,E2 25645.261} C_VEL
LIN {X 0,Y 562.36,Z 882.114,A -85,B 0,C 180,E1 25643.464,E2 25643.464} C_VEL
LIN {X 0,Y 561.757,Z 898.987,A -85,B 0,C 180,E1 25641.605,E2 25641.605} C_VEL
LIN {X 0,Y 561.24,Z 914.727,A -85,B 0,C 180,E1 25639.632,E2 25639.632} C_VEL
LIN {X 0,Y 560.806,Z 929.183,A -85,B 0,C 180,E1 25637.539,E2 25637.539} C_VEL
LIN {X 0,Y 560.474,Z 942.375,A -85,B 0,C 180,E1 25635.324,E2 25635.324} C_VEL
LIN {X 0,Y 560.254,Z 953.3,A -85,B 0,C 180,E1 25633.193,E2 25633.193} C_VEL
LIN {X 0,Y 560.097,Z 963.034,A -85,B 0,C 180,E1 25630.93,E2 25630.93} C_VEL
LIN {X 0,Y 559.99,Z 971.235,A -85,B 0,C 180,E1 25628.637,E2 25628.637} C_VEL
LIN {X 0,Y 559.916,Z 977.465,A -85,B 0,C 180,E1 25626.42,E2 25626.42} C_VEL
LIN {X 0,Y 559.915,Z 982.157,A -85,B 0,C 180,E1 25624.281,E2 25624.281} C_VEL
LIN {X 0,Y 559.91,Z 985.719,A -85,B 0,C 180,E1 25621.87,E2 25621.87} C_VEL
LIN {X 0,Y 559.886,Z 987.564,A -85,B 0,C 180,E1 25619.641,E2 25619.641} C_VEL
LIN {X 0,Y 559.895,Z 987.886,A -85,B 0,C 180,E1 25617.361,E2 25617.361} C_VEL
LIN {X 0,Y 559.914,Z 986.749,A -85,B 0,C 180,E1 25615.023,E2 25615.023} C_VEL
LIN {X 0,Y 559.909,Z 983.796,A -85,B 0,C 180,E1 25612.614,E2 25612.614} C_VEL
LIN {X 0,Y 559.943,Z 979.367,A -85,B 0,C 180,E1 25610.262,E2 25610.262} C_VEL
LIN {X 0,Y 559.961,Z 973.709,A -85,B 0,C 180,E1 25608.1,E2 25608.1} C_VEL
LIN {X 0,Y 560.039,Z 966.214,A -85,B 0,C 180,E1 25605.805,E2 25605.805} C_VEL
LIN {X 0,Y 560.18,Z 957.053,A -85,B 0,C 180,E1 25603.549,E2 25603.549} C_VEL
LIN {X 0,Y 560.4,Z 946.295,A -85,B 0,C 180,E1 25601.309,E2 25601.309} C_VEL
LIN {X 0,Y 560.698,Z 934.014,A -85,B 0,C 180,E1 25599.144,E2 25599.144} C_VEL
LIN {X 0,Y 561.091,Z 919.828,A -85,B 0,C 180,E1 25596.987,E2 25596.987} C_VEL
LIN {X 0,Y 561.58,Z 904.682,A -85,B 0,C 180,E1 25594.981,E2 25594.981} C_VEL
LIN {X 0,Y 562.173,Z 887.691,A -85,B 0,C 180,E1 25593.034,E2 25593.034} C_VEL
LIN {X 0,Y 562.856,Z 869.203,A -85,B 0,C 180,E1 25591.187,E2 25591.187} C_VEL
LIN {X 0,Y 563.595,Z 849.704,A -85,B 0,C 180,E1 25589.493,E2 25589.493} C_VEL
LIN {X 0,Y 564.368,Z 829.64,A -85,B 0,C 180,E1 25588.001,E2 25588.001} C_VEL
LIN {X 0,Y 565.134,Z 808.468,A -85,B 0,C 180,E1 25586.648,E2 25586.648} C_VEL
LIN {X 0,Y 565.899,Z 787.127,A -85,B 0,C 180,E1 25585.503,E2 25585.503} C_VEL
LIN {X 0,Y 566.556,Z 764.429,A -85,B 0,C 180,E1 25584.503,E2 25584.503} C_VEL
LIN {X 0,Y 567.201,Z 741.821,A -85,B 0,C 180,E1 25583.712,E2 25583.712} C_VEL
LIN {X 0,Y 567.625,Z 718.826,A -85,B 0,C 180,E1 25583.113,E2 25583.113} C_VEL
LIN {X 0,Y 567.983,Z 692.683,A -85,B 0,C 180,E1 25582.654,E2 25582.654} C_VEL
LIN {X 0,Y 569.45,Z 481.248,A -85,B 0,C 180,E1 25579.495,E2 25579.495} C_VEL
LIN {X 0,Y 570.065,Z 377.347,A -85,B 0,C 180,E1 25577.888,E2 25577.888} C_VEL
LIN {X 0,Y 563.343,Z 366.707,A -85,B 0,C 180,E1 25577.136,E2 25577.136} C_VEL
LIN {X 0,Y 560.973,Z 363.716,A -85,B 0,C 180,E1 25576.876,E2 25576.876} C_VEL
LIN {X 0,Y 560.345,Z 361.813,A -85,B 0,C 180,E1 25576.749,E2 25576.749} C_VEL
LIN {X 0,Y 560.27,Z 361.26,A -85,B 0,C 180,E1 25576.485,E2 25576.485} C_VEL
LIN {X 0,Y 560.262,Z 361.254,A -85,B 0,C 180,E1 25573.1,E2 25573.1} C_VEL
LIN {X 0,Y 560.269,Z 361.257,A -85,B 0,C 180,E1 25569.865,E2 25569.865} C_VEL
LIN {X 0,Y 560.267,Z 361.26,A -85,B 0,C 180,E1 25566.559,E2 25566.559} C_VEL
LIN {X 0,Y 560.276,Z 361.254,A -85,B 0,C 180,E1 25563.172,E2 25563.172} C_VEL
LIN {X 0,Y 560.263,Z 361.26,A -85,B 0,C 180,E1 25559.796,E2 25559.796} C_VEL
LIN {X 0,Y 560.273,Z 361.256,A -85,B 0,C 180,E1 25556.522,E2 25556.522} C_VEL
LIN {X 0,Y 560.253,Z 361.255,A -85,B 0,C 180,E1 25553.236,E2 25553.236} C_VEL
LIN {X 0,Y 560.266,Z 361.26,A -85,B 0,C 180,E1 25549.824,E2 25549.824} C_VEL
LIN {X 0,Y 560.281,Z 361.255,A -85,B 0,C 180,E1 25546.481,E2 25546.481} C_VEL
LIN {X 0,Y 560.236,Z 361.259,A -85,B 0,C 180,E1 25543.195,E2 25543.195} C_VEL
LIN {X 0,Y 560.281,Z 361.26,A -85,B 0,C 180,E1 25539.963,E2 25539.963} C_VEL
LIN {X 0,Y 560.231,Z 361.258,A -85,B 0,C 180,E1 25536.77,E2 25536.77} C_VEL
LIN {X 0,Y 560.236,Z 361.261,A -85,B 0,C 180,E1 25533.387,E2 25533.387} C_VEL
LIN {X 0,Y 560.25,Z 361.257,A -85,B 0,C 180,E1 25530.256,E2 25530.256} C_VEL
LIN {X 0,Y 560.211,Z 361.263,A -85,B 0,C 180,E1 25527.019,E2 25527.019} C_VEL
LIN {X 0,Y 560.261,Z 361.262,A -85,B 0,C 180,E1 25523.92,E2 25523.92} C_VEL
LIN {X 0,Y 560.196,Z 361.264,A -85,B 0,C 180,E1 25520.683,E2 25520.683} C_VEL
LIN {X 0,Y 560.264,Z 361.259,A -85,B 0,C 180,E1 25517.579,E2 25517.579} C_VEL
LIN {X 0,Y 560.205,Z 361.264,A -85,B 0,C 180,E1 25514.4,E2 25514.4} C_VEL
LIN {X 0,Y 560.321,Z 361.558,A -85,B 0,C 180,E1 25513.489,E2 25513.489} C_VEL
LIN {X 0,Y 561.459,Z 364.6,A -85,B 0,C 180,E1 25513.103,E2 25513.103} C_VEL
LIN {X 0,Y 568.011,Z 378.682,A -85,B 0,C 180,E1 25511.421,E2 25511.421} C_VEL
LIN {X 0,Y 568.239,Z 381.056,A -85,B 0,C 180,E1 25511.222,E2 25511.222} C_VEL
LIN {X 0,Y 568.117,Z 391.551,A -85,B 0,C 180,E1 25510.493,E2 25510.493} C_VEL
LIN {X 0,Y 570.263,Z 402.629,A -85,B 0,C 180,E1 25510.126,E2 25510.126} C_VEL
LIN {X 0,Y 568.756,Z 608.697,A -85,B 0,C 180,E1 25506.991,E2 25506.991} C_VEL
LIN {X 0,Y 567.808,Z 739.997,A -85,B 0,C 180,E1 25505.018,E2 25505.018} C_VEL
LIN {X 0,Y 567.323,Z 763.695,A -85,B 0,C 180,E1 25504.474,E2 25504.474} C_VEL
LIN {X 0,Y 566.851,Z 785.59,A -85,B 0,C 180,E1 25503.785,E2 25503.785} C_VEL
LIN {X 0,Y 566.167,Z 807.65,A -85,B 0,C 180,E1 25502.893,E2 25502.893} C_VEL
LIN {X 0,Y 565.506,Z 828.755,A -85,B 0,C 180,E1 25501.857,E2 25501.857} C_VEL
LIN {X 0,Y 564.724,Z 849.819,A -85,B 0,C 180,E1 25500.607,E2 25500.607} C_VEL
LIN {X 0,Y 563.961,Z 870.382,A -85,B 0,C 180,E1 25499.182,E2 25499.182} C_VEL
LIN {X 0,Y 563.25,Z 888.567,A -85,B 0,C 180,E1 25497.718,E2 25497.718} C_VEL
LIN {X 0,Y 562.524,Z 907.961,A -85,B 0,C 180,E1 25495.923,E2 25495.923} C_VEL
LIN {X 0,Y 561.904,Z 925.171,A -85,B 0,C 180,E1 25494.101,E2 25494.101} C_VEL
LIN {X 0,Y 561.36,Z 941.097,A -85,B 0,C 180,E1 25492.152,E2 25492.152} C_VEL
LIN {X 0,Y 560.902,Z 956.322,A -85,B 0,C 180,E1 25490.017,E2 25490.017} C_VEL
LIN {X 0,Y 560.561,Z 968.994,A -85,B 0,C 180,E1 25487.976,E2 25487.976} C_VEL
LIN {X 0,Y 560.298,Z 980.308,A -85,B 0,C 180,E1 25485.847,E2 25485.847} C_VEL
LIN {X 0,Y 560.126,Z 989.986,A -85,B 0,C 180,E1 25483.736,E2 25483.736} C_VEL
LIN {X 0,Y 560.022,Z 998.332,A -85,B 0,C 180,E1 25481.537,E2 25481.537} C_VEL
LIN {X 0,Y 559.945,Z 1004.862,A -85,B 0,C 180,E1 25479.458,E2 25479.458} C_VEL
LIN {X 0,Y 559.898,Z 1010.629,A -85,B 0,C 180,E1 25477.08,E2 25477.08} C_VEL
LIN {X 0,Y 559.91,Z 1014.272,A -85,B 0,C 180,E1 25475.022,E2 25475.022} C_VEL
LIN {X 0,Y 559.914,Z 1016.986,A -85,B 0,C 180,E1 25472.561,E2 25472.561} C_VEL
LIN {X 0,Y 559.887,Z 1017.916,A -85,B 0,C 180,E1 25470.412,E2 25470.412} C_VEL
LIN {X 0,Y 559.914,Z 1017.326,A -85,B 0,C 180,E1 25467.956,E2 25467.956} C_VEL
LIN {X 0,Y 559.909,Z 1015.279,A -85,B 0,C 180,E1 25465.702,E2 25465.702} C_VEL
LIN {X 0,Y 559.914,Z 1011.466,A -85,B 0,C 180,E1 25463.337,E2 25463.337} C_VEL
LIN {X 0,Y 559.951,Z 1006.558,A -85,B 0,C 180,E1 25461.17,E2 25461.17} C_VEL
LIN {X 0,Y 559.989,Z 999.775,A -85,B 0,C 180,E1 25458.885,E2 25458.885} C_VEL
LIN {X 0,Y 560.098,Z 992.122,A -85,B 0,C 180,E1 25456.795,E2 25456.795} C_VEL
LIN {X 0,Y 560.275,Z 981.899,A -85,B 0,C 180,E1 25454.477,E2 25454.477} C_VEL
LIN {X 0,Y 560.529,Z 970.839,A -85,B 0,C 180,E1 25452.351,E2 25452.351} C_VEL
LIN {X 0,Y 560.856,Z 957.777,A -85,B 0,C 180,E1 25450.205,E2 25450.205} C_VEL
LIN {X 0,Y 561.289,Z 943.348,A -85,B 0,C 180,E1 25448.138,E2 25448.138} C_VEL
LIN {X 0,Y 561.805,Z 927.975,A -85,B 0,C 180,E1 25446.231,E2 25446.231} C_VEL
LIN {X 0,Y 562.436,Z 910.155,A -85,B 0,C 180,E1 25444.297,E2 25444.297} C_VEL
LIN {X 0,Y 563.119,Z 892.256,A -85,B 0,C 180,E1 25442.595,E2 25442.595} C_VEL
LIN {X 0,Y 563.841,Z 873.393,A -85,B 0,C 180,E1 25441.05,E2 25441.05} C_VEL
LIN {X 0,Y 564.607,Z 852.67,A -85,B 0,C 180,E1 25439.575,E2 25439.575} C_VEL
LIN {X 0,Y 565.351,Z 832.907,A -85,B 0,C 180,E1 25438.378,E2 25438.378} C_VEL
LIN {X 0,Y 566.073,Z 810.172,A -85,B 0,C 180,E1 25437.22,E2 25437.22} C_VEL
LIN {X 0,Y 566.758,Z 788.881,A -85,B 0,C 180,E1 25436.336,E2 25436.336} C_VEL
LIN {X 0,Y 567.282,Z 766.019,A -85,B 0,C 180,E1 25435.591,E2 25435.591} C_VEL
LIN {X 0,Y 567.767,Z 743.523,A -85,B 0,C 180,E1 25435.045,E2 25435.045} C_VEL
LIN {X 0,Y 568.125,Z 701.487,A -85,B 0,C 180,E1 25434.387,E2 25434.387} C_VEL
LIN {X 0,Y 569.581,Z 492.325,A -85,B 0,C 180,E1 25431.251,E2 25431.251} C_VEL
LIN {X 0,Y 570.119,Z 401.012,A -85,B 0,C 180,E1 25429.836,E2 25429.836} C_VEL
LIN {X 0,Y 568.014,Z 390.66,A -85,B 0,C 180,E1 25429.465,E2 25429.465} C_VEL
LIN {X 0,Y 568.218,Z 379.137,A -85,B 0,C 180,E1 25428.632,E2 25428.632} C_VEL
LIN {X 0,Y 562.876,Z 367.723,A -85,B 0,C 180,E1 25427.274,E2 25427.274} C_VEL
LIN {X 0,Y 560.325,Z 361.565,A -85,B 0,C 180,E1 25426.515,E2 25426.515} C_VEL
LIN {X 0,Y 560.205,Z 361.254,A -85,B 0,C 180,E1 25425.409,E2 25425.409} C_VEL
LIN {X 0,Y 560.27,Z 361.251,A -85,B 0,C 180,E1 25422.223,E2 25422.223} C_VEL
LIN {X 0,Y 560.2,Z 361.251,A -85,B 0,C 180,E1 25419.185,E2 25419.185} C_VEL
LIN {X 0,Y 560.267,Z 361.248,A -85,B 0,C 180,E1 25416.065,E2 25416.065} C_VEL
LIN {X 0,Y 560.197,Z 361.263,A -85,B 0,C 180,E1 25412.981,E2 25412.981} C_VEL
LIN {X 0,Y 560.245,Z 361.251,A -85,B 0,C 180,E1 25409.745,E2 25409.745} C_VEL
LIN {X 0,Y 560.194,Z 361.263,A -85,B 0,C 180,E1 25406.729,E2 25406.729} C_VEL
LIN {X 0,Y 560.232,Z 361.259,A -85,B 0,C 180,E1 25403.452,E2 25403.452} C_VEL
LIN {X 0,Y 560.202,Z 361.261,A -85,B 0,C 180,E1 25400.476,E2 25400.476} C_VEL
LIN {X 0,Y 560.223,Z 361.26,A -85,B 0,C 180,E1 25397.126,E2 25397.126} C_VEL
LIN {X 0,Y 560.216,Z 361.26,A -85,B 0,C 180,E1 25394.153,E2 25394.153} C_VEL
LIN {X 0,Y 560.216,Z 361.259,A -85,B 0,C 180,E1 25390.801,E2 25390.801} C_VEL
LIN {X 0,Y 560.235,Z 361.26,A -85,B 0,C 180,E1 25387.795,E2 25387.795} C_VEL
LIN {X 0,Y 560.215,Z 361.257,A -85,B 0,C 180,E1 25384.504,E2 25384.504} C_VEL
LIN {X 0,Y 560.273,Z 361.258,A -85,B 0,C 180,E1 25381.329,E2 25381.329} C_VEL
LIN {X 0,Y 560.215,Z 361.257,A -85,B 0,C 180,E1 25378.159,E2 25378.159} C_VEL
LIN {X 0,Y 560.282,Z 361.255,A -85,B 0,C 180,E1 25374.983,E2 25374.983} C_VEL
LIN {X 0,Y 560.221,Z 361.259,A -85,B 0,C 180,E1 25371.791,E2 25371.791} C_VEL
LIN {X 0,Y 560.276,Z 361.255,A -85,B 0,C 180,E1 25368.574,E2 25368.574} C_VEL
LIN {X 0,Y 560.231,Z 361.259,A -85,B 0,C 180,E1 25365.425,E2 25365.425} C_VEL
LIN {X 0,Y 560.243,Z 361.256,A -85,B 0,C 180,E1 25362.016,E2 25362.016} C_VEL
LIN {X 0,Y 560.275,Z 361.259,A -85,B 0,C 180,E1 25358.76,E2 25358.76} C_VEL
LIN {X 0,Y 560.28,Z 361.253,A -85,B 0,C 180,E1 25356.235,E2 25356.235} C_VEL
LIN {X 0,Y 559.256,Z 361.379,A -85,B 0,C 180,E1 25355.447,E2 25355.447} C_VEL
LIN {X 0,Y 552.826,Z 362.185,A -85,B 0,C 180,E1 25353.236,E2 25353.236} C_VEL
LIN {X 0,Y 552.332,Z 362.246,A -85,B 0,C 180,E1 25352.66,E2 25352.66} C_VEL
LIN {X 0,Y 552.299,Z 362.243,A -85,B 0,C 180,E1 25349.299,E2 25349.299} C_VEL
LIN {X 0,Y 552.342,Z 362.242,A -85,B 0,C 180,E1 25345.988,E2 25345.988} C_VEL
LIN {X 0,Y 552.312,Z 362.248,A -85,B 0,C 180,E1 25342.666,E2 25342.666} C_VEL
LIN {X 0,Y 552.317,Z 362.24,A -85,B 0,C 180,E1 25339.327,E2 25339.327} C_VEL
LIN {X 0,Y 552.342,Z 362.246,A -85,B 0,C 180,E1 25335.963,E2 25335.963} C_VEL
LIN {X 0,Y 552.309,Z 362.243,A -85,B 0,C 180,E1 25332.693,E2 25332.693} C_VEL
LIN {X 0,Y 552.343,Z 362.241,A -85,B 0,C 180,E1 25329.309,E2 25329.309} C_VEL
LIN {X 0,Y 552.34,Z 362.25,A -85,B 0,C 180,E1 25325.905,E2 25325.905} C_VEL
LIN {X 0,Y 552.314,Z 362.246,A -85,B 0,C 180,E1 25322.52,E2 25322.52} C_VEL
LIN {X 0,Y 552.336,Z 362.243,A -85,B 0,C 180,E1 25319.245,E2 25319.245} C_VEL
LIN {X 0,Y 552.331,Z 362.237,A -85,B 0,C 180,E1 25315.862,E2 25315.862} C_VEL
LIN {X 0,Y 552.325,Z 362.243,A -85,B 0,C 180,E1 25312.452,E2 25312.452} C_VEL
LIN {X 0,Y 552.331,Z 362.246,A -85,B 0,C 180,E1 25309.099,E2 25309.099} C_VEL
LIN {X 0,Y 552.327,Z 362.247,A -85,B 0,C 180,E1 25305.753,E2 25305.753} C_VEL
LIN {X 0,Y 552.335,Z 362.214,A -85,B 0,C 180,E1 25302.331,E2 25302.331} C_VEL
LIN {X 0,Y 552.361,Z 362.485,A -85,B 0,C 180,E1 25299.952,E2 25299.952} C_VEL
LIN {X 0,Y 552.736,Z 363.95,A -85,B 0,C 180,E1 25299.778,E2 25299.778} C_VEL
LIN {X 0,Y 554.736,Z 366.998,A -85,B 0,C 180,E1 25299.542,E2 25299.542} C_VEL
LIN {X 0,Y 555.9,Z 368.66,A -85,B 0,C 180,E1 25299.407,E2 25299.407} C_VEL
LIN {X 0,Y 564.066,Z 381.104,A -85,B 0,C 180,E1 25298.474,E2 25298.474} C_VEL
LIN {X 0,Y 562.278,Z 589.355,A -85,B 0,C 180,E1 25295.277,E2 25295.277} C_VEL
LIN {X 0,Y 561.246,Z 710.971,A -85,B 0,C 180,E1 25293.428,E2 25293.428} C_VEL
LIN {X 0,Y 560.679,Z 734.796,A -85,B 0,C 180,E1 25292.869,E2 25292.869} C_VEL
LIN {X 0,Y 560.04,Z 758.542,A -85,B 0,C 180,E1 25292.095,E2 25292.095} C_VEL
LIN {X 0,Y 559.235,Z 780.489,A -85,B 0,C 180,E1 25291.175,E2 25291.175} C_VEL
LIN {X 0,Y 558.367,Z 803.342,A -85,B 0,C 180,E1 25289.997,E2 25289.997} C_VEL
LIN {X 0,Y 557.447,Z 824.153,A -85,B 0,C 180,E1 25288.713,E2 25288.713} C_VEL
LIN {X 0,Y 556.564,Z 844.265,A -85,B 0,C 180,E1 25287.252,E2 25287.252} C_VEL
LIN {X 0,Y 555.645,Z 864.391,A -85,B 0,C 180,E1 25285.56,E2 25285.56} C_VEL
LIN {X 0,Y 554.82,Z 882.87,A -85,B 0,C 180,E1 25283.755,E2 25283.755} C_VEL
LIN {X 0,Y 554.115,Z 899.361,A -85,B 0,C 180,E1 25281.907,E2 25281.907} C_VEL
LIN {X 0,Y 553.497,Z 915.063,A -85,B 0,C 180,E1 25279.903,E2 25279.903} C_VEL
LIN {X 0,Y 552.995,Z 929.463,A -85,B 0,C 180,E1 25277.785,E2 25277.785} C_VEL
LIN {X 0,Y 552.594,Z 942.598,A -85,B 0,C 180,E1 25275.538,E2 25275.538} C_VEL
LIN {X 0,Y 552.315,Z 954.018,A -85,B 0,C 180,E1 25273.267,E2 25273.267} C_VEL
LIN {X 0,Y 552.127,Z 963.646,A -85,B 0,C 180,E1 25270.962,E2 25270.962} C_VEL
LIN {X 0,Y 552.004,Z 971.855,A -85,B 0,C 180,E1 25268.595,E2 25268.595} C_VEL
LIN {X 0,Y 551.921,Z 977.821,A -85,B 0,C 180,E1 25266.397,E2 25266.397} C_VEL
LIN {X 0,Y 551.904,Z 982.637,A -85,B 0,C 180,E1 25264.11,E2 25264.11} C_VEL
LIN {X 0,Y 551.912,Z 985.971,A -85,B 0,C 180,E1 25261.697,E2 25261.697} C_VEL
LIN {X 0,Y 551.904,Z 987.71,A -85,B 0,C 180,E1 25259.377,E2 25259.377} C_VEL
LIN {X 0,Y 551.903,Z 987.828,A -85,B 0,C 180,E1 25257.076,E2 25257.076} C_VEL
LIN {X 0,Y 551.91,Z 986.356,A -85,B 0,C 180,E1 25254.567,E2 25254.567} C_VEL
LIN {X 0,Y 551.893,Z 983.25,A -85,B 0,C 180,E1 25252.176,E2 25252.176} C_VEL
LIN {X 0,Y 551.924,Z 978.614,A -85,B 0,C 180,E1 25249.838,E2 25249.838} C_VEL
LIN {X 0,Y 551.988,Z 973.187,A -85,B 0,C 180,E1 25247.775,E2 25247.775} C_VEL
LIN {X 0,Y 552.083,Z 965.215,A -85,B 0,C 180,E1 25245.355,E2 25245.355} C_VEL
LIN {X 0,Y 552.25,Z 956.211,A -85,B 0,C 180,E1 25243.142,E2 25243.142} C_VEL
LIN {X 0,Y 552.523,Z 944.843,A -85,B 0,C 180,E1 25240.789,E2 25240.789} C_VEL
LIN {X 0,Y 552.895,Z 932.444,A -85,B 0,C 180,E1 25238.602,E2 25238.602} C_VEL
LIN {X 0,Y 553.378,Z 918.382,A -85,B 0,C 180,E1 25236.474,E2 25236.474} C_VEL
LIN {X 0,Y 553.985,Z 902.646,A -85,B 0,C 180,E1 25234.397,E2 25234.397} C_VEL
LIN {X 0,Y 554.702,Z 885.511,A -85,B 0,C 180,E1 25232.429,E2 25232.429} C_VEL
LIN {X 0,Y 555.52,Z 867.306,A -85,B 0,C 180,E1 25230.622,E2 25230.622} C_VEL
LIN {X 0,Y 556.415,Z 847.439,A -85,B 0,C 180,E1 25228.907,E2 25228.907} C_VEL
LIN {X 0,Y 557.293,Z 827.981,A -85,B 0,C 180,E1 25227.458,E2 25227.458} C_VEL
LIN {X 0,Y 558.185,Z 807.368,A -85,B 0,C 180,E1 25226.146,E2 25226.146} C_VEL
LIN {X 0,Y 559.029,Z 786.545,A -85,B 0,C 180,E1 25225.024,E2 25225.024} C_VEL
LIN {X 0,Y 559.816,Z 764.085,A -85,B 0,C 180,E1 25224.031,E2 25224.031} C_VEL
LIN {X 0,Y 560.539,Z 741.644,A -85,B 0,C 180,E1 25223.242,E2 25223.242} C_VEL
LIN {X 0,Y 561.058,Z 718.23,A -85,B 0,C 180,E1 25222.63,E2 25222.63} C_VEL
LIN {X 0,Y 561.467,Z 690.815,A -85,B 0,C 180,E1 25222.153,E2 25222.153} C_VEL
LIN {X 0,Y 563.2,Z 479.425,A -85,B 0,C 180,E1 25218.959,E2 25218.959} C_VEL
LIN {X 0,Y 563.964,Z 380.834,A -85,B 0,C 180,E1 25217.422,E2 25217.422} C_VEL
LIN {X 0,Y 557.488,Z 371.237,A -85,B 0,C 180,E1 25216.69,E2 25216.69} C_VEL
LIN {X 0,Y 554.853,Z 367.118,A -85,B 0,C 180,E1 25216.381,E2 25216.381} C_VEL
LIN {X 0,Y 552.775,Z 364.011,A -85,B 0,C 180,E1 25216.136,E2 25216.136} C_VEL
LIN {X 0,Y 552.403,Z 362.669,A -85,B 0,C 180,E1 25216.006,E2 25216.006} C_VEL
LIN {X 0,Y 552.338,Z 362.199,A -85,B 0,C 180,E1 25215.54,E2 25215.54} C_VEL
LIN {X 0,Y 552.338,Z 362.246,A -85,B 0,C 180,E1 25212.122,E2 25212.122} C_VEL
LIN {X 0,Y 552.324,Z 362.249,A -85,B 0,C 180,E1 25208.727,E2 25208.727} C_VEL
LIN {X 0,Y 552.335,Z 362.244,A -85,B 0,C 180,E1 25205.351,E2 25205.351} C_VEL
LIN {X 0,Y 552.327,Z 362.249,A -85,B 0,C 180,E1 25201.868,E2 25201.868} C_VEL
LIN {X 0,Y 552.334,Z 362.246,A -85,B 0,C 180,E1 25198.548,E2 25198.548} C_VEL
LIN {X 0,Y 552.318,Z 362.241,A -85,B 0,C 180,E1 25195.224,E2 25195.224} C_VEL
LIN {X 0,Y 552.323,Z 362.25,A -85,B 0,C 180,E1 25191.778,E2 25191.778} C_VEL
LIN {X 0,Y 552.342,Z 362.244,A -85,B 0,C 180,E1 25188.409,E2 25188.409} C_VEL
LIN {X 0,Y 552.301,Z 362.246,A -85,B 0,C 180,E1 25185.104,E2 25185.104} C_VEL
LIN {X 0,Y 552.326,Z 362.25,A -85,B 0,C 180,E1 25181.75,E2 25181.75} C_VEL
LIN {X 0,Y 552.317,Z 362.246,A -85,B 0,C 180,E1 25178.514,E2 25178.514} C_VEL
LIN {X 0,Y 552.286,Z 362.25,A -85,B 0,C 180,E1 25175.165,E2 25175.165} C_VEL
LIN {X 0,Y 552.345,Z 362.248,A -85,B 0,C 180,E1 25171.924,E2 25171.924} C_VEL
LIN {X 0,Y 552.272,Z 362.25,A -85,B 0,C 180,E1 25168.817,E2 25168.817} C_VEL
LIN {X 0,Y 552.323,Z 362.248,A -85,B 0,C 180,E1 25165.612,E2 25165.612} C_VEL
LIN {X 0,Y 552.266,Z 362.252,A -85,B 0,C 180,E1 25162.467,E2 25162.467} C_VEL
LIN {X 0,Y 552.269,Z 362.254,A -85,B 0,C 180,E1 25159.024,E2 25159.024} C_VEL
LIN {X 0,Y 552.293,Z 362.247,A -85,B 0,C 180,E1 25155.951,E2 25155.951} C_VEL
LIN {X 0,Y 552.309,Z 362.5,A -85,B 0,C 180,E1 25154.202,E2 25154.202} C_VEL
LIN {X 0,Y 553.713,Z 365.863,A -85,B 0,C 180,E1 25153.756,E2 25153.756} C_VEL
LIN {X 0,Y 561.707,Z 383.072,A -85,B 0,C 180,E1 25151.655,E2 25151.655} C_VEL
LIN {X 0,Y 561.645,Z 391.667,A -85,B 0,C 180,E1 25151.057,E2 25151.057} C_VEL
LIN {X 0,Y 564.128,Z 404.37,A -85,B 0,C 180,E1 25150.625,E2 25150.625} C_VEL
LIN {X 0,Y 562.348,Z 610.606,A -85,B 0,C 180,E1 25147.454,E2 25147.454} C_VEL
LIN {X 0,Y 561.248,Z 739.996,A -85,B 0,C 180,E1 25145.489,E2 25145.489} C_VEL
LIN {X 0,Y 560.696,Z 763.693,A -85,B 0,C 180,E1 25144.941,E2 25144.941} C_VEL
LIN {X 0,Y 560.123,Z 785.615,A -85,B 0,C 180,E1 25144.246,E2 25144.246} C_VEL
LIN {X 0,Y 559.345,Z 807.647,A -85,B 0,C 180,E1 25143.346,E2 25143.346} C_VEL
LIN {X 0,Y 558.545,Z 828.755,A -85,B 0,C 180,E1 25142.302,E2 25142.302} C_VEL
LIN {X 0,Y 557.683,Z 849.022,A -85,B 0,C 180,E1 25141.09,E2 25141.09} C_VEL
LIN {X 0,Y 556.797,Z 868.91,A -85,B 0,C 180,E1 25139.713,E2 25139.713} C_VEL
LIN {X 0,Y 555.951,Z 887.508,A -85,B 0,C 180,E1 25138.208,E2 25138.208} C_VEL
LIN {X 0,Y 555.08,Z 906.775,A -85,B 0,C 180,E1 25136.42,E2 25136.42} C_VEL
LIN {X 0,Y 554.356,Z 923.645,A -85,B 0,C 180,E1 25134.625,E2 25134.625} C_VEL
LIN {X 0,Y 553.689,Z 939.979,A -85,B 0,C 180,E1 25132.623,E2 25132.623} C_VEL
LIN {X 0,Y 553.14,Z 954.907,A -85,B 0,C 180,E1 25130.531,E2 25130.531} C_VEL
LIN {X 0,Y 552.723,Z 967.722,A -85,B 0,C 180,E1 25128.458,E2 25128.458} C_VEL
LIN {X 0,Y 552.398,Z 979.788,A -85,B 0,C 180,E1 25126.188,E2 25126.188} C_VEL
LIN {X 0,Y 552.192,Z 989.526,A -85,B 0,C 180,E1 25124.044,E2 25124.044} C_VEL
LIN {X 0,Y 552.053,Z 998.333,A -85,B 0,C 180,E1 25121.706,E2 25121.706} C_VEL
LIN {X 0,Y 551.954,Z 1005.165,A -85,B 0,C 180,E1 25119.491,E2 25119.491} C_VEL
LIN {X 0,Y 551.902,Z 1010.629,A -85,B 0,C 180,E1 25117.183,E2 25117.183} C_VEL
LIN {X 0,Y 551.913,Z 1014.273,A -85,B 0,C 180,E1 25115.095,E2 25115.095} C_VEL
LIN {X 0,Y 551.911,Z 1016.986,A -85,B 0,C 180,E1 25112.598,E2 25112.598} C_VEL
LIN {X 0,Y 551.884,Z 1017.894,A -85,B 0,C 180,E1 25110.522,E2 25110.522} C_VEL
LIN {X 0,Y 551.911,Z 1017.393,A -85,B 0,C 180,E1 25108.03,E2 25108.03} C_VEL
LIN {X 0,Y 551.914,Z 1015.506,A -85,B 0,C 180,E1 25105.847,E2 25105.847} C_VEL
LIN {X 0,Y 551.918,Z 1011.673,A -85,B 0,C 180,E1 25103.345,E2 25103.345} C_VEL
LIN {X 0,Y 551.953,Z 1007.069,A -85,B 0,C 180,E1 25101.251,E2 25101.251} C_VEL
LIN {X 0,Y 552.008,Z 1000.13,A -85,B 0,C 180,E1 25098.828,E2 25098.828} C_VEL
LIN {X 0,Y 552.13,Z 992.532,A -85,B 0,C 180,E1 25096.707,E2 25096.707} C_VEL
LIN {X 0,Y 552.34,Z 982.417,A -85,B 0,C 180,E1 25094.356,E2 25094.356} C_VEL
LIN {X 0,Y 552.619,Z 972.001,A -85,B 0,C 180,E1 25092.308,E2 25092.308} C_VEL
LIN {X 0,Y 553.032,Z 958.488,A -85,B 0,C 180,E1 25090.023,E2 25090.023} C_VEL
LIN {X 0,Y 553.548,Z 944.073,A -85,B 0,C 180,E1 25087.912,E2 25087.912} C_VEL
LIN {X 0,Y 554.169,Z 928.239,A -85,B 0,C 180,E1 25085.915,E2 25085.915} C_VEL
LIN {X 0,Y 554.943,Z 910.156,A -85,B 0,C 180,E1 25083.924,E2 25083.924} C_VEL
LIN {X 0,Y 555.761,Z 891.944,A -85,B 0,C 180,E1 25082.173,E2 25082.173} C_VEL
LIN {X 0,Y 556.616,Z 872.911,A -85,B 0,C 180,E1 25080.599,E2 25080.599} C_VEL
LIN {X 0,Y 557.556,Z 851.784,A -85,B 0,C 180,E1 25079.089,E2 25079.089} C_VEL
LIN {X 0,Y 558.372,Z 832.904,A -85,B 0,C 180,E1 25077.936,E2 25077.936} C_VEL
LIN {X 0,Y 559.244,Z 809.984,A -85,B 0,C 180,E1 25076.759,E2 25076.759} C_VEL
LIN {X 0,Y 560.023,Z 788.879,A -85,B 0,C 180,E1 25075.876,E2 25075.876} C_VEL
LIN {X 0,Y 560.634,Z 765.955,A -85,B 0,C 180,E1 25075.123,E2 25075.123} C_VEL
LIN {X 0,Y 561.212,Z 743.179,A -85,B 0,C 180,E1 25074.568,E2 25074.568} C_VEL
LIN {X 0,Y 561.66,Z 696.788,A -85,B 0,C 180,E1 25073.84,E2 25073.84} C_VEL
LIN {X 0,Y 563.366,Z 488.89,A -85,B 0,C 180,E1 25070.687,E2 25070.687} C_VEL
LIN {X 0,Y 563.983,Z 402.785,A -85,B 0,C 180,E1 25069.337,E2 25069.337} C_VEL
LIN {X 0,Y 561.522,Z 390.884,A -85,B 0,C 180,E1 25068.911,E2 25068.911} C_VEL
LIN {X 0,Y 561.609,Z 382.833,A -85,B 0,C 180,E1 25068.318,E2 25068.318} C_VEL
LIN {X 0,Y 553.716,Z 365.855,A -85,B 0,C 180,E1 25066.243,E2 25066.243} C_VEL
LIN {X 0,Y 552.316,Z 362.511,A -85,B 0,C 180,E1 25065.797,E2 25065.797} C_VEL
LIN {X 0,Y 552.267,Z 362.228,A -85,B 0,C 180,E1 25063.152,E2 25063.152} C_VEL
LIN {X 0,Y 552.292,Z 362.235,A -85,B 0,C 180,E1 25059.857,E2 25059.857} C_VEL
LIN {X 0,Y 552.273,Z 362.253,A -85,B 0,C 180,E1 25056.816,E2 25056.816} C_VEL
LIN {X 0,Y 552.266,Z 362.252,A -85,B 0,C 180,E1 25053.393,E2 25053.393} C_VEL
LIN {X 0,Y 552.281,Z 362.239,A -85,B 0,C 180,E1 25050.458,E2 25050.458} C_VEL
LIN {X 0,Y 552.258,Z 362.252,A -85,B 0,C 180,E1 25047.145,E2 25047.145} C_VEL
LIN {X 0,Y 552.309,Z 362.252,A -85,B 0,C 180,E1 25044.036,E2 25044.036} C_VEL
LIN {X 0,Y 552.261,Z 362.25,A -85,B 0,C 180,E1 25040.895,E2 25040.895} C_VEL
LIN {X 0,Y 552.33,Z 362.248,A -85,B 0,C 180,E1 25037.705,E2 25037.705} C_VEL
LIN {X 0,Y 552.262,Z 362.248,A -85,B 0,C 180,E1 25034.575,E2 25034.575} C_VEL
LIN {X 0,Y 552.337,Z 362.245,A -85,B 0,C 180,E1 25031.38,E2 25031.38} C_VEL
LIN {X 0,Y 552.27,Z 362.248,A -85,B 0,C 180,E1 25028.223,E2 25028.223} C_VEL
LIN {X 0,Y 552.316,Z 362.244,A -85,B 0,C 180,E1 25024.985,E2 25024.985} C_VEL
LIN {X 0,Y 552.282,Z 362.249,A -85,B 0,C 180,E1 25021.867,E2 25021.867} C_VEL
LIN {X 0,Y 552.288,Z 362.246,A -85,B 0,C 180,E1 25018.444,E2 25018.444} C_VEL
LIN {X 0,Y 552.317,Z 362.251,A -85,B 0,C 180,E1 25015.327,E2 25015.327} C_VEL
LIN {X 0,Y 552.284,Z 362.247,A -85,B 0,C 180,E1 25012.091,E2 25012.091} C_VEL
LIN {X 0,Y 552.345,Z 362.247,A -85,B 0,C 180,E1 25008.827,E2 25008.827} C_VEL
LIN {X 0,Y 552.289,Z 362.248,A -85,B 0,C 180,E1 25005.532,E2 25005.532} C_VEL
LIN {X 0,Y 552.318,Z 362.245,A -85,B 0,C 180,E1 25002.185,E2 25002.185} C_VEL
LIN {X 0,Y 552.315,Z 362.246,A -85,B 0,C 180,E1 24998.995,E2 24998.995} C_VEL
LIN {X 0,Y 552.295,Z 362.245,A -85,B 0,C 180,E1 24995.621,E2 24995.621} C_VEL
LIN {X 0,Y 552.332,Z 362.246,A -85,B 0,C 180,E1 24992.66,E2 24992.66} C_VEL
LIN {X 0,Y 551.374,Z 362.368,A -85,B 0,C 180,E1 24991.861,E2 24991.861} C_VEL
LIN {X 0,Y 544.882,Z 363.167,A -85,B 0,C 180,E1 24989.617,E2 24989.617} C_VEL
LIN {X 0,Y 544.362,Z 363.233,A -85,B 0,C 180,E1 24989.032,E2 24989.032} C_VEL
LIN {X 0,Y 544.385,Z 363.23,A -85,B 0,C 180,E1 24985.677,E2 24985.677} C_VEL
LIN {X 0,Y 544.401,Z 363.234,A -85,B 0,C 180,E1 24982.295,E2 24982.295} C_VEL
LIN {X 0,Y 544.366,Z 363.23,A -85,B 0,C 180,E1 24979.01,E2 24979.01} C_VEL
LIN {X 0,Y 544.402,Z 363.233,A -85,B 0,C 180,E1 24975.74,E2 24975.74} C_VEL
LIN {X 0,Y 544.382,Z 363.234,A -85,B 0,C 180,E1 24972.376,E2 24972.376} C_VEL
LIN {X 0,Y 544.377,Z 363.233,A -85,B 0,C 180,E1 24968.909,E2 24968.909} C_VEL
LIN {X 0,Y 544.399,Z 363.233,A -85,B 0,C 180,E1 24965.548,E2 24965.548} C_VEL
LIN {X 0,Y 544.383,Z 363.238,A -85,B 0,C 180,E1 24962.179,E2 24962.179} C_VEL
LIN {X 0,Y 544.391,Z 363.231,A -85,B 0,C 180,E1 24958.76,E2 24958.76} C_VEL
LIN {X 0,Y 544.394,Z 363.224,A -85,B 0,C 180,E1 24955.36,E2 24955.36} C_VEL
LIN {X 0,Y 544.383,Z 363.23,A -85,B 0,C 180,E1 24952.001,E2 24952.001} C_VEL
LIN {X 0,Y 544.4,Z 363.23,A -85,B 0,C 180,E1 24948.612,E2 24948.612} C_VEL
LIN {X 0,Y 544.395,Z 363.234,A -85,B 0,C 180,E1 24945.223,E2 24945.223} C_VEL
LIN {X 0,Y 544.384,Z 363.206,A -85,B 0,C 180,E1 24941.868,E2 24941.868} C_VEL
LIN {X 0,Y 544.435,Z 363.546,A -85,B 0,C 180,E1 24940.686,E2 24940.686} C_VEL
LIN {X 0,Y 544.893,Z 365.177,A -85,B 0,C 180,E1 24940.499,E2 24940.499} C_VEL
LIN {X 0,Y 546.911,Z 368.112,A -85,B 0,C 180,E1 24940.254,E2 24940.254} C_VEL
LIN {X 0,Y 548.137,Z 369.93,A -85,B 0,C 180,E1 24940.106,E2 24940.106} C_VEL
LIN {X 0,Y 557.948,Z 384.511,A -85,B 0,C 180,E1 24938.957,E2 24938.957} C_VEL
LIN {X 0,Y 555.873,Z 593.749,A -85,B 0,C 180,E1 24935.712,E2 24935.712} C_VEL
LIN {X 0,Y 554.72,Z 711.036,A -85,B 0,C 180,E1 24933.908,E2 24933.908} C_VEL
LIN {X 0,Y 554.088,Z 734.805,A -85,B 0,C 180,E1 24933.346,E2 24933.346} C_VEL
LIN {X 0,Y 553.338,Z 758.693,A -85,B 0,C 180,E1 24932.56,E2 24932.56} C_VEL
LIN {X 0,Y 552.456,Z 780.102,A -85,B 0,C 180,E1 24931.657,E2 24931.657} C_VEL
LIN {X 0,Y 551.477,Z 802.215,A -85,B 0,C 180,E1 24930.517,E2 24930.517} C_VEL
LIN {X 0,Y 550.431,Z 823.162,A -85,B 0,C 180,E1 24929.217,E2 24929.217} C_VEL
LIN {X 0,Y 549.358,Z 843.932,A -85,B 0,C 180,E1 24927.703,E2 24927.703} C_VEL
LIN {X 0,Y 548.318,Z 863.71,A -85,B 0,C 180,E1 24926.024,E2 24926.024} C_VEL
LIN {X 0,Y 547.36,Z 882.413,A -85,B 0,C 180,E1 24924.182,E2 24924.182} C_VEL
LIN {X 0,Y 546.486,Z 899.735,A -85,B 0,C 180,E1 24922.216,E2 24922.216} C_VEL
LIN {X 0,Y 545.735,Z 916.123,A -85,B 0,C 180,E1 24920.081,E2 24920.081} C_VEL
LIN {X 0,Y 545.137,Z 930.894,A -85,B 0,C 180,E1 24917.85,E2 24917.85} C_VEL
LIN {X 0,Y 544.674,Z 943.977,A -85,B 0,C 180,E1 24915.541,E2 24915.541} C_VEL
LIN {X 0,Y 544.338,Z 955.62,A -85,B 0,C 180,E1 24913.127,E2 24913.127} C_VEL
LIN {X 0,Y 544.149,Z 964.595,A -85,B 0,C 180,E1 24910.907,E2 24910.907} C_VEL
LIN {X 0,Y 544.015,Z 972.774,A -85,B 0,C 180,E1 24908.431,E2 24908.431} C_VEL
LIN {X 0,Y 543.927,Z 978.453,A -85,B 0,C 180,E1 24906.259,E2 24906.259} C_VEL
LIN {X 0,Y 543.895,Z 983.255,A -85,B 0,C 180,E1 24903.818,E2 24903.818} C_VEL
LIN {X 0,Y 543.909,Z 986.301,A -85,B 0,C 180,E1 24901.446,E2 24901.446} C_VEL
LIN {X 0,Y 543.91,Z 987.818,A -85,B 0,C 180,E1 24898.896,E2 24898.896} C_VEL
LIN {X 0,Y 543.905,Z 987.725,A -85,B 0,C 180,E1 24896.573,E2 24896.573} C_VEL
LIN {X 0,Y 543.912,Z 985.98,A -85,B 0,C 180,E1 24894.163,E2 24894.163} C_VEL
LIN {X 0,Y 543.903,Z 982.87,A -85,B 0,C 180,E1 24891.852,E2 24891.852} C_VEL
LIN {X 0,Y 543.926,Z 978.188,A -85,B 0,C 180,E1 24889.54,E2 24889.54} C_VEL
LIN {X 0,Y 544.013,Z 972.661,A -85,B 0,C 180,E1 24887.438,E2 24887.438} C_VEL
LIN {X 0,Y 544.153,Z 964.478,A -85,B 0,C 180,E1 24884.973,E2 24884.973} C_VEL
LIN {X 0,Y 544.348,Z 955.321,A -85,B 0,C 180,E1 24882.715,E2 24882.715} C_VEL
LIN {X 0,Y 544.673,Z 944.001,A -85,B 0,C 180,E1 24880.373,E2 24880.373} C_VEL
LIN {X 0,Y 545.123,Z 931.169,A -85,B 0,C 180,E1 24878.105,E2 24878.105} C_VEL
LIN {X 0,Y 545.713,Z 916.592,A -85,B 0,C 180,E1 24875.896,E2 24875.896} C_VEL
LIN {X 0,Y 546.481,Z 899.89,A -85,B 0,C 180,E1 24873.712,E2 24873.712} C_VEL
LIN {X 0,Y 547.351,Z 882.56,A -85,B 0,C 180,E1 24871.742,E2 24871.742} C_VEL
LIN {X 0,Y 548.296,Z 864.06,A -85,B 0,C 180,E1 24869.918,E2 24869.918} C_VEL
LIN {X 0,Y 549.337,Z 844.368,A -85,B 0,C 180,E1 24868.243,E2 24868.243} C_VEL
LIN {X 0,Y 550.416,Z 823.45,A -85,B 0,C 180,E1 24866.712,E2 24866.712} C_VEL
LIN {X 0,Y 551.435,Z 803.128,A -85,B 0,C 180,E1 24865.447,E2 24865.447} C_VEL
LIN {X 0,Y 552.419,Z 780.848,A -85,B 0,C 180,E1 24864.288,E2 24864.288} C_VEL
LIN {X 0,Y 553.325,Z 759.207,A -85,B 0,C 180,E1 24863.369,E2 24863.369} C_VEL
LIN {X 0,Y 554.074,Z 735.272,A -85,B 0,C 180,E1 24862.577,E2 24862.577} C_VEL
LIN {X 0,Y 554.704,Z 711.789,A -85,B 0,C 180,E1 24862.016,E2 24862.016} C_VEL
LIN {X 0,Y 555.364,Z 648.209,A -85,B 0,C 180,E1 24861.026,E2 24861.026} C_VEL
LIN {X 0,Y 557.39,Z 438.803,A -85,B 0,C 180,E1 24857.806,E2 24857.806} C_VEL
LIN {X 0,Y 557.795,Z 384.239,A -85,B 0,C 180,E1 24856.935,E2 24856.935} C_VEL
LIN {X 0,Y 549.541,Z 372.108,A -85,B 0,C 180,E1 24855.974,E2 24855.974} C_VEL
LIN {X 0,Y 547.025,Z 368.19,A -85,B 0,C 180,E1 24855.668,E2 24855.668} C_VEL
LIN {X 0,Y 544.893,Z 365.142,A -85,B 0,C 180,E1 24855.41,E2 24855.41} C_VEL
LIN {X 0,Y 544.487,Z 363.813,A -85,B 0,C 180,E1 24855.282,E2 24855.282} C_VEL
LIN {X 0,Y 544.373,Z 363.185,A -85,B 0,C 180,E1 24854.956,E2 24854.956} C_VEL
LIN {X 0,Y 544.395,Z 363.229,A -85,B 0,C 180,E1 24851.656,E2 24851.656} C_VEL
LIN {X 0,Y 544.401,Z 363.235,A -85,B 0,C 180,E1 24848.237,E2 24848.237} C_VEL
LIN {X 0,Y 544.391,Z 363.235,A -85,B 0,C 180,E1 24844.847,E2 24844.847} C_VEL
LIN {X 0,Y 544.384,Z 363.235,A -85,B 0,C 180,E1 24841.474,E2 24841.474} C_VEL
LIN {X 0,Y 544.4,Z 363.235,A -85,B 0,C 180,E1 24838.106,E2 24838.106} C_VEL
LIN {X 0,Y 544.4,Z 363.229,A -85,B 0,C 180,E1 24834.626,E2 24834.626} C_VEL
LIN {X 0,Y 544.371,Z 363.236,A -85,B 0,C 180,E1 24831.338,E2 24831.338} C_VEL
LIN {X 0,Y 544.4,Z 363.238,A -85,B 0,C 180,E1 24828.022,E2 24828.022} C_VEL
LIN {X 0,Y 544.391,Z 363.232,A -85,B 0,C 180,E1 24824.635,E2 24824.635} C_VEL
LIN {X 0,Y 544.356,Z 363.237,A -85,B 0,C 180,E1 24821.251,E2 24821.251} C_VEL
LIN {X 0,Y 544.408,Z 363.237,A -85,B 0,C 180,E1 24817.997,E2 24817.997} C_VEL
LIN {X 0,Y 544.35,Z 363.238,A -85,B 0,C 180,E1 24814.778,E2 24814.778} C_VEL
LIN {X 0,Y 544.355,Z 363.237,A -85,B 0,C 180,E1 24811.354,E2 24811.354} C_VEL
LIN {X 0,Y 544.363,Z 363.239,A -85,B 0,C 180,E1 24808.259,E2 24808.259} C_VEL
LIN {X 0,Y 544.332,Z 363.242,A -85,B 0,C 180,E1 24805.01,E2 24805.01} C_VEL
LIN {X 0,Y 544.39,Z 363.238,A -85,B 0,C 180,E1 24801.761,E2 24801.761} C_VEL
LIN {X 0,Y 544.318,Z 363.245,A -85,B 0,C 180,E1 24798.545,E2 24798.545} C_VEL
LIN {X 0,Y 544.369,Z 363.226,A -85,B 0,C 180,E1 24795.295,E2 24795.295} C_VEL
LIN {X 0,Y 544.375,Z 363.512,A -85,B 0,C 180,E1 24794.885,E2 24794.885} C_VEL
LIN {X 0,Y 545.935,Z 367.16,A -85,B 0,C 180,E1 24794.398,E2 24794.398} C_VEL
LIN {X 0,Y 555.178,Z 386.848,A -85,B 0,C 180,E1 24791.964,E2 24791.964} C_VEL
LIN {X 0,Y 555.203,Z 391.689,A -85,B 0,C 180,E1 24791.638,E2 24791.638} C_VEL
LIN {X 0,Y 558.035,Z 406.271,A -85,B 0,C 180,E1 24791.132,E2 24791.132} C_VEL
LIN {X 0,Y 555.978,Z 612.514,A -85,B 0,C 180,E1 24787.928,E2 24787.928} C_VEL
LIN {X 0,Y 554.726,Z 740.176,A -85,B 0,C 180,E1 24785.967,E2 24785.967} C_VEL
LIN {X 0,Y 554.108,Z 763.692,A -85,B 0,C 180,E1 24785.418,E2 24785.418} C_VEL
LIN {X 0,Y 553.435,Z 785.474,A -85,B 0,C 180,E1 24784.724,E2 24784.724} C_VEL
LIN {X 0,Y 552.6,Z 806.764,A -85,B 0,C 180,E1 24783.851,E2 24783.851} C_VEL
LIN {X 0,Y 551.716,Z 826.529,A -85,B 0,C 180,E1 24782.875,E2 24782.875} C_VEL
LIN {X 0,Y 550.687,Z 848.033,A -85,B 0,C 180,E1 24781.597,E2 24781.597} C_VEL
LIN {X 0,Y 549.67,Z 868.165,A -85,B 0,C 180,E1 24780.198,E2 24780.198} C_VEL
LIN {X 0,Y 548.622,Z 887.865,A -85,B 0,C 180,E1 24778.587,E2 24778.587} C_VEL
LIN {X 0,Y 547.596,Z 907.197,A -85,B 0,C 180,E1 24776.765,E2 24776.765} C_VEL
LIN {X 0,Y 546.746,Z 924.655,A -85,B 0,C 180,E1 24774.875,E2 24774.875} C_VEL
LIN {X 0,Y 545.97,Z 940.827,A -85,B 0,C 180,E1 24772.847,E2 24772.847} C_VEL
LIN {X 0,Y 545.305,Z 956.326,A -85,B 0,C 180,E1 24770.615,E2 24770.615} C_VEL
LIN {X 0,Y 544.835,Z 968.99,A -85,B 0,C 180,E1 24768.513,E2 24768.513} C_VEL
LIN {X 0,Y 544.477,Z 980.311,A -85,B 0,C 180,E1 24766.32,E2 24766.32} C_VEL
LIN {X 0,Y 544.227,Z 990.442,A -85,B 0,C 180,E1 24764.037,E2 24764.037} C_VEL
LIN {X 0,Y 544.074,Z 998.69,A -85,B 0,C 180,E1 24761.773,E2 24761.773} C_VEL
LIN {X 0,Y 543.965,Z 1005.768,A -85,B 0,C 180,E1 24759.418,E2 24759.418} C_VEL
LIN {X 0,Y 543.905,Z 1010.836,A -85,B 0,C 180,E1 24757.184,E2 24757.184} C_VEL
LIN {X 0,Y 543.913,Z 1014.432,A -85,B 0,C 180,E1 24755.065,E2 24755.065} C_VEL
LIN {X 0,Y 543.913,Z 1017.054,A -85,B 0,C 180,E1 24752.531,E2 24752.531} C_VEL
LIN {X 0,Y 543.892,Z 1017.939,A -85,B 0,C 180,E1 24750.319,E2 24750.319} C_VEL
LIN {X 0,Y 543.914,Z 1017.326,A -85,B 0,C 180,E1 24747.896,E2 24747.896} C_VEL
LIN {X 0,Y 543.908,Z 1015.393,A -85,B 0,C 180,E1 24745.68,E2 24745.68} C_VEL
LIN {X 0,Y 543.915,Z 1011.673,A -85,B 0,C 180,E1 24743.247,E2 24743.247} C_VEL
LIN {X 0,Y 543.964,Z 1007.069,A -85,B 0,C 180,E1 24741.121,E2 24741.121} C_VEL
LIN {X 0,Y 544.033,Z 1000.129,A -85,B 0,C 180,E1 24738.662,E2 24738.662} C_VEL
LIN {X 0,Y 544.17,Z 992.533,A -85,B 0,C 180,E1 24736.509,E2 24736.509} C_VEL
LIN {X 0,Y 544.419,Z 982.416,A -85,B 0,C 180,E1 24734.122,E2 24734.122} C_VEL
LIN {X 0,Y 544.746,Z 972.003,A -85,B 0,C 180,E1 24732.043,E2 24732.043} C_VEL
LIN {X 0,Y 545.234,Z 958.488,A -85,B 0,C 180,E1 24729.725,E2 24729.725} C_VEL
LIN {X 0,Y 545.837,Z 944.245,A -85,B 0,C 180,E1 24727.607,E2 24727.607} C_VEL
LIN {X 0,Y 546.545,Z 928.441,A -85,B 0,C 180,E1 24725.582,E2 24725.582} C_VEL
LIN {X 0,Y 547.463,Z 910.156,A -85,B 0,C 180,E1 24723.541,E2 24723.541} C_VEL
LIN {X 0,Y 548.427,Z 891.946,A -85,B 0,C 180,E1 24721.768,E2 24721.768} C_VEL
LIN {X 0,Y 549.41,Z 872.653,A -85,B 0,C 180,E1 24720.154,E2 24720.154} C_VEL
LIN {X 0,Y 550.535,Z 851.112,A -85,B 0,C 180,E1 24718.604,E2 24718.604} C_VEL
LIN {X 0,Y 551.471,Z 831.896,A -85,B 0,C 180,E1 24717.424,E2 24717.424} C_VEL
LIN {X 0,Y 552.434,Z 810.335,A -85,B 0,C 180,E1 24716.312,E2 24716.312} C_VEL
LIN {X 0,Y 553.252,Z 790.496,A -85,B 0,C 180,E1 24715.468,E2 24715.468} C_VEL
LIN {X 0,Y 554.002,Z 767.048,A -85,B 0,C 180,E1 24714.676,E2 24714.676} C_VEL
LIN {X 0,Y 554.608,Z 745.308,A -85,B 0,C 180,E1 24714.133,E2 24714.133} C_VEL
LIN {X 0,Y 555.058,Z 712.183,A -85,B 0,C 180,E1 24713.584,E2 24713.584} C_VEL
LIN {X 0,Y 557.062,Z 501.385,A -85,B 0,C 180,E1 24710.359,E2 24710.359} C_VEL
LIN {X 0,Y 557.889,Z 404.571,A -85,B 0,C 180,E1 24708.827,E2 24708.827} C_VEL
LIN {X 0,Y 555.076,Z 390.452,A -85,B 0,C 180,E1 24708.3,E2 24708.3} C_VEL
LIN {X 0,Y 555.036,Z 386.483,A -85,B 0,C 180,E1 24707.995,E2 24707.995} C_VEL
LIN {X 0,Y 547.079,Z 369.769,A -85,B 0,C 180,E1 24705.91,E2 24705.91} C_VEL
LIN {X 0,Y 544.393,Z 363.603,A -85,B 0,C 180,E1 24705.113,E2 24705.113} C_VEL
LIN {X 0,Y 544.387,Z 363.198,A -85,B 0,C 180,E1 24704.556,E2 24704.556} C_VEL
LIN {X 0,Y 544.327,Z 363.244,A -85,B 0,C 180,E1 24701.305,E2 24701.305} C_VEL
LIN {X 0,Y 544.378,Z 363.234,A -85,B 0,C 180,E1 24698.013,E2 24698.013} C_VEL
LIN {X 0,Y 544.327,Z 363.221,A -85,B 0,C 180,E1 24694.815,E2 24694.815} C_VEL
LIN {X 0,Y 544.325,Z 363.233,A -85,B 0,C 180,E1 24691.321,E2 24691.321} C_VEL
LIN {X 0,Y 544.35,Z 363.235,A -85,B 0,C 180,E1 24688.287,E2 24688.287} C_VEL
LIN {X 0,Y 544.318,Z 363.241,A -85,B 0,C 180,E1 24684.991,E2 24684.991} C_VEL
LIN {X 0,Y 544.399,Z 363.238,A -85,B 0,C 180,E1 24681.777,E2 24681.777} C_VEL
LIN {X 0,Y 544.324,Z 363.24,A -85,B 0,C 180,E1 24678.528,E2 24678.528} C_VEL
LIN {X 0,Y 544.363,Z 363.237,A -85,B 0,C 180,E1 24675.227,E2 24675.227} C_VEL
LIN {X 0,Y 544.334,Z 363.24,A -85,B 0,C 180,E1 24672.195,E2 24672.195} C_VEL
LIN {X 0,Y 544.343,Z 363.236,A -85,B 0,C 180,E1 24668.769,E2 24668.769} C_VEL
LIN {X 0,Y 544.364,Z 363.24,A -85,B 0,C 180,E1 24665.692,E2 24665.692} C_VEL
LIN {X 0,Y 544.337,Z 363.237,A -85,B 0,C 180,E1 24662.356,E2 24662.356} C_VEL
LIN {X 0,Y 544.405,Z 363.236,A -85,B 0,C 180,E1 24659.158,E2 24659.158} C_VEL
LIN {X 0,Y 544.342,Z 363.238,A -85,B 0,C 180,E1 24655.892,E2 24655.892} C_VEL
LIN {X 0,Y 544.385,Z 363.235,A -85,B 0,C 180,E1 24652.613,E2 24652.613} C_VEL
LIN {X 0,Y 544.36,Z 363.237,A -85,B 0,C 180,E1 24649.416,E2 24649.416} C_VEL
LIN {X 0,Y 544.352,Z 363.235,A -85,B 0,C 180,E1 24645.968,E2 24645.968} C_VEL
LIN {X 0,Y 544.405,Z 363.236,A -85,B 0,C 180,E1 24642.69,E2 24642.69} C_VEL
LIN {X 0,Y 544.353,Z 363.232,A -85,B 0,C 180,E1 24639.462,E2 24639.462} C_VEL
LIN {X 0,Y 544.394,Z 363.231,A -85,B 0,C 180,E1 24636.144,E2 24636.144} C_VEL
LIN {X 0,Y 544.372,Z 363.237,A -85,B 0,C 180,E1 24632.902,E2 24632.902} C_VEL
LIN {X 0,Y 544.363,Z 363.231,A -85,B 0,C 180,E1 24629.469,E2 24629.469} C_VEL
LIN {X 0,Y 544.362,Z 363.233,A -85,B 0,C 180,E1 24629.032,E2 24629.032} C_VEL
LIN {X 0,Y 543.404,Z 363.36,A -85,B 0,C 180,E1 24628.221,E2 24628.221} C_VEL
LIN {X 0,Y 536.88,Z 364.167,A -85,B 0,C 180,E1 24625.885,E2 24625.885} C_VEL
LIN {X 0,Y 536.427,Z 364.221,A -85,B 0,C 180,E1 24625.35,E2 24625.35} C_VEL
LIN {X 0,Y 536.465,Z 364.224,A -85,B 0,C 180,E1 24622.027,E2 24622.027} C_VEL
LIN {X 0,Y 536.433,Z 364.221,A -85,B 0,C 180,E1 24618.684,E2 24618.684} C_VEL
LIN {X 0,Y 536.441,Z 364.221,A -85,B 0,C 180,E1 24615.207,E2 24615.207} C_VEL
LIN {X 0,Y 536.463,Z 364.224,A -85,B 0,C 180,E1 24611.796,E2 24611.796} C_VEL
LIN {X 0,Y 536.436,Z 364.225,A -85,B 0,C 180,E1 24608.479,E2 24608.479} C_VEL
LIN {X 0,Y 536.455,Z 364.219,A -85,B 0,C 180,E1 24605.029,E2 24605.029} C_VEL
LIN {X 0,Y 536.458,Z 364.212,A -85,B 0,C 180,E1 24601.578,E2 24601.578} C_VEL
LIN {X 0,Y 536.44,Z 364.224,A -85,B 0,C 180,E1 24598.253,E2 24598.253} C_VEL
LIN {X 0,Y 536.459,Z 364.216,A -85,B 0,C 180,E1 24594.79,E2 24594.79} C_VEL
LIN {X 0,Y 536.459,Z 364.209,A -85,B 0,C 180,E1 24591.423,E2 24591.423} C_VEL
LIN {X 0,Y 536.444,Z 364.216,A -85,B 0,C 180,E1 24588.02,E2 24588.02} C_VEL
LIN {X 0,Y 536.463,Z 364.21,A -85,B 0,C 180,E1 24584.57,E2 24584.57} C_VEL
LIN {X 0,Y 536.474,Z 364.349,A -85,B 0,C 180,E1 24581.5,E2 24581.5} C_VEL
LIN {X 0,Y 536.852,Z 365.879,A -85,B 0,C 180,E1 24581.288,E2 24581.288} C_VEL
LIN {X 0,Y 538.869,Z 369.02,A -85,B 0,C 180,E1 24581.023,E2 24581.023} C_VEL
LIN {X 0,Y 540.067,Z 370.546,A -85,B 0,C 180,E1 24580.876,E2 24580.876} C_VEL
LIN {X 0,Y 551.868,Z 388.16,A -85,B 0,C 180,E1 24579.446,E2 24579.446} C_VEL
LIN {X 0,Y 549.494,Z 598.775,A -85,B 0,C 180,E1 24576.147,E2 24576.147} C_VEL
LIN {X 0,Y 548.24,Z 710.931,A -85,B 0,C 180,E1 24574.403,E2 24574.403} C_VEL
LIN {X 0,Y 547.545,Z 734.688,A -85,B 0,C 180,E1 24573.838,E2 24573.838} C_VEL
LIN {X 0,Y 546.685,Z 758.463,A -85,B 0,C 180,E1 24573.052,E2 24573.052} C_VEL
LIN {X 0,Y 545.72,Z 779.71,A -85,B 0,C 180,E1 24572.15,E2 24572.15} C_VEL
LIN {X 0,Y 544.577,Z 801.957,A -85,B 0,C 180,E1 24570.997,E2 24570.997} C_VEL
LIN {X 0,Y 543.457,Z 822.173,A -85,B 0,C 180,E1 24569.734,E2 24569.734} C_VEL
LIN {X 0,Y 542.199,Z 843.384,A -85,B 0,C 180,E1 24568.182,E2 24568.182} C_VEL
LIN {X 0,Y 541.036,Z 863.024,A -85,B 0,C 180,E1 24566.501,E2 24566.501} C_VEL
LIN {X 0,Y 539.92,Z 881.862,A -85,B 0,C 180,E1 24564.632,E2 24564.632} C_VEL
LIN {X 0,Y 538.914,Z 899.237,A -85,B 0,C 180,E1 24562.642,E2 24562.642} C_VEL
LIN {X 0,Y 538.107,Z 914.91,A -85,B 0,C 180,E1 24560.587,E2 24560.587} C_VEL
LIN {X 0,Y 537.427,Z 929.335,A -85,B 0,C 180,E1 24558.406,E2 24558.406} C_VEL
LIN {X 0,Y 536.869,Z 942.471,A -85,B 0,C 180,E1 24556.096,E2 24556.096} C_VEL
LIN {X 0,Y 536.488,Z 953.867,A -85,B 0,C 180,E1 24553.764,E2 24553.764} C_VEL
LIN {X 0,Y 536.219,Z 963.472,A -85,B 0,C 180,E1 24551.404,E2 24551.404} C_VEL
LIN {X 0,Y 536.041,Z 971.564,A -85,B 0,C 180,E1 24549.012,E2 24549.012} C_VEL
LIN {X 0,Y 535.946,Z 977.706,A -85,B 0,C 180,E1 24546.7,E2 24546.7} C_VEL
LIN {X 0,Y 535.92,Z 982.613,A -85,B 0,C 180,E1 24544.307,E2 24544.307} C_VEL
LIN {X 0,Y 535.906,Z 985.834,A -85,B 0,C 180,E1 24541.945,E2 24541.945} C_VEL
LIN {X 0,Y 535.892,Z 987.655,A -85,B 0,C 180,E1 24539.541,E2 24539.541} C_VEL
LIN {X 0,Y 535.897,Z 987.87,A -85,B 0,C 180,E1 24537.241,E2 24537.241} C_VEL
LIN {X 0,Y 535.913,Z 986.655,A -85,B 0,C 180,E1 24534.793,E2 24534.793} C_VEL
LIN {X 0,Y 535.9,Z 983.846,A -85,B 0,C 180,E1 24532.401,E2 24532.401} C_VEL
LIN {X 0,Y 535.947,Z 979.679,A -85,B 0,C 180,E1 24530.064,E2 24530.064} C_VEL
LIN {X 0,Y 536.016,Z 973.755,A -85,B 0,C 180,E1 24527.669,E2 24527.669} C_VEL
LIN {X 0,Y 536.136,Z 966.294,A -85,B 0,C 180,E1 24525.279,E2 24525.279} C_VEL
LIN {X 0,Y 536.364,Z 957.054,A -85,B 0,C 180,E1 24522.893,E2 24522.893} C_VEL
LIN {X 0,Y 536.72,Z 946.172,A -85,B 0,C 180,E1 24520.528,E2 24520.528} C_VEL
LIN {X 0,Y 537.203,Z 933.734,A -85,B 0,C 180,E1 24518.237,E2 24518.237} C_VEL
LIN {X 0,Y 537.866,Z 919.425,A -85,B 0,C 180,E1 24515.975,E2 24515.975} C_VEL
LIN {X 0,Y 538.684,Z 903.855,A -85,B 0,C 180,E1 24513.837,E2 24513.837} C_VEL
LIN {X 0,Y 539.636,Z 886.681,A -85,B 0,C 180,E1 24511.798,E2 24511.798} C_VEL
LIN {X 0,Y 540.688,Z 868.801,A -85,B 0,C 180,E1 24509.954,E2 24509.954} C_VEL
LIN {X 0,Y 541.893,Z 849.081,A -85,B 0,C 180,E1 24508.187,E2 24508.187} C_VEL
LIN {X 0,Y 543.046,Z 828.878,A -85,B 0,C 180,E1 24506.637,E2 24506.637} C_VEL
LIN {X 0,Y 544.251,Z 808.249,A -85,B 0,C 180,E1 24505.286,E2 24505.286} C_VEL
LIN {X 0,Y 545.378,Z 786.241,A -85,B 0,C 180,E1 24504.075,E2 24504.075} C_VEL
LIN {X 0,Y 546.43,Z 764.114,A -85,B 0,C 180,E1 24503.082,E2 24503.082} C_VEL
LIN {X 0,Y 547.31,Z 742.286,A -85,B 0,C 180,E1 24502.298,E2 24502.298} C_VEL
LIN {X 0,Y 548.016,Z 718.441,A -85,B 0,C 180,E1 24501.662,E2 24501.662} C_VEL
LIN {X 0,Y 548.519,Z 691.877,A -85,B 0,C 180,E1 24501.189,E2 24501.189} C_VEL
LIN {X 0,Y 550.796,Z 480.728,A -85,B 0,C 180,E1 24497.928,E2 24497.928} C_VEL
LIN {X 0,Y 551.761,Z 387.787,A -85,B 0,C 180,E1 24496.448,E2 24496.448} C_VEL
LIN {X 0,Y 542.034,Z 373.569,A -85,B 0,C 180,E1 24495.281,E2 24495.281} C_VEL
LIN {X 0,Y 539.297,Z 369.369,A -85,B 0,C 180,E1 24494.934,E2 24494.934} C_VEL
LIN {X 0,Y 537.051,Z 366.401,A -85,B 0,C 180,E1 24494.653,E2 24494.653} C_VEL
LIN {X 0,Y 536.532,Z 364.71,A -85,B 0,C 180,E1 24494.489,E2 24494.489} C_VEL
LIN {X 0,Y 536.456,Z 364.175,A -85,B 0,C 180,E1 24494.133,E2 24494.133} C_VEL
LIN {X 0,Y 536.443,Z 364.211,A -85,B 0,C 180,E1 24490.742,E2 24490.742} C_VEL
LIN {X 0,Y 536.466,Z 364.222,A -85,B 0,C 180,E1 24487.281,E2 24487.281} C_VEL
LIN {X 0,Y 536.451,Z 364.227,A -85,B 0,C 180,E1 24483.848,E2 24483.848} C_VEL
LIN {X 0,Y 536.455,Z 364.226,A -85,B 0,C 180,E1 24480.428,E2 24480.428} C_VEL
LIN {X 0,Y 536.456,Z 364.22,A -85,B 0,C 180,E1 24477.009,E2 24477.009} C_VEL
LIN {X 0,Y 536.437,Z 364.225,A -85,B 0,C 180,E1 24473.579,E2 24473.579} C_VEL
LIN {X 0,Y 536.462,Z 364.225,A -85,B 0,C 180,E1 24470.235,E2 24470.235} C_VEL
LIN {X 0,Y 536.44,Z 364.223,A -85,B 0,C 180,E1 24466.857,E2 24466.857} C_VEL
LIN {X 0,Y 536.425,Z 364.228,A -85,B 0,C 180,E1 24463.431,E2 24463.431} C_VEL
LIN {X 0,Y 536.467,Z 364.225,A -85,B 0,C 180,E1 24460.058,E2 24460.058} C_VEL
LIN {X 0,Y 536.415,Z 364.226,A -85,B 0,C 180,E1 24456.773,E2 24456.773} C_VEL
LIN {X 0,Y 536.415,Z 364.229,A -85,B 0,C 180,E1 24453.307,E2 24453.307} C_VEL
LIN {X 0,Y 536.459,Z 364.221,A -85,B 0,C 180,E1 24450.033,E2 24450.033} C_VEL
LIN {X 0,Y 536.392,Z 364.23,A -85,B 0,C 180,E1 24446.769,E2 24446.769} C_VEL
LIN {X 0,Y 536.427,Z 364.226,A -85,B 0,C 180,E1 24443.453,E2 24443.453} C_VEL
LIN {X 0,Y 536.393,Z 364.233,A -85,B 0,C 180,E1 24440.256,E2 24440.256} C_VEL
LIN {X 0,Y 536.386,Z 364.236,A -85,B 0,C 180,E1 24436.792,E2 24436.792} C_VEL
LIN {X 0,Y 536.482,Z 364.434,A -85,B 0,C 180,E1 24435.62,E2 24435.62} C_VEL
LIN {X 0,Y 537.656,Z 367.598,A -85,B 0,C 180,E1 24435.186,E2 24435.186} C_VEL
LIN {X 0,Y 546.614,Z 386.301,A -85,B 0,C 180,E1 24432.82,E2 24432.82} C_VEL
LIN {X 0,Y 548.711,Z 391.154,A -85,B 0,C 180,E1 24432.254,E2 24432.254} C_VEL
LIN {X 0,Y 551.988,Z 408.051,A -85,B 0,C 180,E1 24431.652,E2 24431.652} C_VEL
LIN {X 0,Y 549.643,Z 614.805,A -85,B 0,C 180,E1 24428.407,E2 24428.407} C_VEL
LIN {X 0,Y 548.241,Z 740.363,A -85,B 0,C 180,E1 24426.457,E2 24426.457} C_VEL
LIN {X 0,Y 547.557,Z 763.82,A -85,B 0,C 180,E1 24425.903,E2 24425.903} C_VEL
LIN {X 0,Y 546.777,Z 785.803,A -85,B 0,C 180,E1 24425.197,E2 24425.197} C_VEL
LIN {X 0,Y 545.818,Z 807.482,A -85,B 0,C 180,E1 24424.294,E2 24424.294} C_VEL
LIN {X 0,Y 544.809,Z 827.651,A -85,B 0,C 180,E1 24423.282,E2 24423.282} C_VEL
LIN {X 0,Y 543.656,Z 848.472,A -85,B 0,C 180,E1 24422.023,E2 24422.023} C_VEL
LIN {X 0,Y 542.487,Z 868.904,A -85,B 0,C 180,E1 24420.579,E2 24420.579} C_VEL
LIN {X 0,Y 541.331,Z 887.911,A -85,B 0,C 180,E1 24419.004,E2 24419.004} C_VEL
LIN {X 0,Y 540.172,Z 907.157,A -85,B 0,C 180,E1 24417.167,E2 24417.167} C_VEL
LIN {X 0,Y 539.219,Z 924.271,A -85,B 0,C 180,E1 24415.291,E2 24415.291} C_VEL
LIN {X 0,Y 538.34,Z 939.98,A -85,B 0,C 180,E1 24413.306,E2 24413.306} C_VEL
LIN {X 0,Y 537.604,Z 954.91,A -85,B 0,C 180,E1 24411.152,E2 24411.152} C_VEL
LIN {X 0,Y 537.052,Z 967.718,A -85,B 0,C 180,E1 24409.017,E2 24409.017} C_VEL
LIN {X 0,Y 536.601,Z 979.791,A -85,B 0,C 180,E1 24406.678,E2 24406.678} C_VEL
LIN {X 0,Y 536.318,Z 989.523,A -85,B 0,C 180,E1 24404.469,E2 24404.469} C_VEL
LIN {X 0,Y 536.106,Z 998.335,A -85,B 0,C 180,E1 24402.059,E2 24402.059} C_VEL
LIN {X 0,Y 535.972,Z 1005.164,A -85,B 0,C 180,E1 24399.776,E2 24399.776} C_VEL
LIN {X 0,Y 535.916,Z 1010.629,A -85,B 0,C 180,E1 24397.399,E2 24397.399} C_VEL
LIN {X 0,Y 535.916,Z 1014.273,A -85,B 0,C 180,E1 24395.248,E2 24395.248} C_VEL
LIN {X 0,Y 535.905,Z 1016.986,A -85,B 0,C 180,E1 24392.676,E2 24392.676} C_VEL
LIN {X 0,Y 535.885,Z 1017.894,A -85,B 0,C 180,E1 24390.537,E2 24390.537} C_VEL
LIN {X 0,Y 535.913,Z 1017.393,A -85,B 0,C 180,E1 24387.971,E2 24387.971} C_VEL
LIN {X 0,Y 535.91,Z 1015.506,A -85,B 0,C 180,E1 24385.723,E2 24385.723} C_VEL
LIN {X 0,Y 535.909,Z 1011.673,A -85,B 0,C 180,E1 24383.145,E2 24383.145} C_VEL
LIN {X 0,Y 535.976,Z 1007.069,A -85,B 0,C 180,E1 24380.988,E2 24380.988} C_VEL
LIN {X 0,Y 536.065,Z 1000.128,A -85,B 0,C 180,E1 24378.491,E2 24378.491} C_VEL
LIN {X 0,Y 536.218,Z 992.448,A -85,B 0,C 180,E1 24376.282,E2 24376.282} C_VEL
LIN {X 0,Y 536.507,Z 982.414,A -85,B 0,C 180,E1 24373.882,E2 24373.882} C_VEL
LIN {X 0,Y 536.872,Z 971.998,A -85,B 0,C 180,E1 24371.769,E2 24371.769} C_VEL
LIN {X 0,Y 537.442,Z 958.486,A -85,B 0,C 180,E1 24369.418,E2 24369.418} C_VEL
LIN {X 0,Y 538.144,Z 944.245,A -85,B 0,C 180,E1 24367.27,E2 24367.27} C_VEL
LIN {X 0,Y 538.953,Z 928.441,A -85,B 0,C 180,E1 24365.215,E2 24365.215} C_VEL
LIN {X 0,Y 540.002,Z 910.157,A -85,B 0,C 180,E1 24363.146,E2 24363.146} C_VEL
LIN {X 0,Y 541.109,Z 892.1,A -85,B 0,C 180,E1 24361.366,E2 24361.366} C_VEL
LIN {X 0,Y 542.227,Z 872.65,A -85,B 0,C 180,E1 24359.718,E2 24359.718} C_VEL
LIN {X 0,Y 543.472,Z 851.965,A -85,B 0,C 180,E1 24358.208,E2 24358.208} C_VEL
LIN {X 0,Y 544.512,Z 832.898,A -85,B 0,C 180,E1 24357.018,E2 24357.018} C_VEL
LIN {X 0,Y 545.677,Z 810.339,A -85,B 0,C 180,E1 24355.838,E2 24355.838} C_VEL
LIN {X 0,Y 546.558,Z 791.094,A -85,B 0,C 180,E1 24355.01,E2 24355.01} C_VEL
LIN {X 0,Y 547.413,Z 767.871,A -85,B 0,C 180,E1 24354.212,E2 24354.212} C_VEL
LIN {X 0,Y 548.074,Z 746.443,A -85,B 0,C 180,E1 24353.666,E2 24353.666} C_VEL
LIN {X 0,Y 548.589,Z 715.188,A -85,B 0,C 180,E1 24353.132,E2 24353.132} C_VEL
LIN {X 0,Y 550.856,Z 505.179,A -85,B 0,C 180,E1 24349.886,E2 24349.886} C_VEL
LIN {X 0,Y 551.835,Z 406.346,A -85,B 0,C 180,E1 24348.305,E2 24348.305} C_VEL
LIN {X 0,Y 548.672,Z 390.704,A -85,B 0,C 180,E1 24347.719,E2 24347.719} C_VEL
LIN {X 0,Y 540.179,Z 372.549,A -85,B 0,C 180,E1 24345.448,E2 24345.448} C_VEL
LIN {X 0,Y 536.536,Z 364.683,A -85,B 0,C 180,E1 24344.395,E2 24344.395} C_VEL
LIN {X 0,Y 536.416,Z 364.183,A -85,B 0,C 180,E1 24343.994,E2 24343.994} C_VEL
LIN {X 0,Y 536.406,Z 364.226,A -85,B 0,C 180,E1 24340.825,E2 24340.825} C_VEL
LIN {X 0,Y 536.39,Z 364.232,A -85,B 0,C 180,E1 24337.422,E2 24337.422} C_VEL
LIN {X 0,Y 536.45,Z 364.21,A -85,B 0,C 180,E1 24334.126,E2 24334.126} C_VEL
LIN {X 0,Y 536.38,Z 364.22,A -85,B 0,C 180,E1 24330.963,E2 24330.963} C_VEL
LIN {X 0,Y 536.43,Z 364.23,A -85,B 0,C 180,E1 24327.714,E2 24327.714} C_VEL
LIN {X 0,Y 536.386,Z 364.23,A -85,B 0,C 180,E1 24324.552,E2 24324.552} C_VEL
LIN {X 0,Y 536.392,Z 364.228,A -85,B 0,C 180,E1 24321.085,E2 24321.085} C_VEL
LIN {X 0,Y 536.43,Z 364.23,A -85,B 0,C 180,E1 24317.911,E2 24317.911} C_VEL
LIN {X 0,Y 536.388,Z 364.226,A -85,B 0,C 180,E1 24314.679,E2 24314.679} C_VEL
LIN {X 0,Y 536.456,Z 364.223,A -85,B 0,C 180,E1 24311.503,E2 24311.503} C_VEL
LIN {X 0,Y 536.393,Z 364.226,A -85,B 0,C 180,E1 24308.222,E2 24308.222} C_VEL
LIN {X 0,Y 536.431,Z 364.222,A -85,B 0,C 180,E1 24304.918,E2 24304.918} C_VEL
LIN {X 0,Y 536.417,Z 364.228,A -85,B 0,C 180,E1 24301.709,E2 24301.709} C_VEL
LIN {X 0,Y 536.403,Z 364.224,A -85,B 0,C 180,E1 24298.291,E2 24298.291} C_VEL
LIN {X 0,Y 536.465,Z 364.221,A -85,B 0,C 180,E1 24294.974,E2 24294.974} C_VEL
LIN {X 0,Y 536.407,Z 364.227,A -85,B 0,C 180,E1 24291.748,E2 24291.748} C_VEL
LIN {X 0,Y 536.437,Z 364.223,A -85,B 0,C 180,E1 24288.387,E2 24288.387} C_VEL
LIN {X 0,Y 536.442,Z 364.228,A -85,B 0,C 180,E1 24285.095,E2 24285.095} C_VEL
LIN {X 0,Y 536.414,Z 364.225,A -85,B 0,C 180,E1 24281.751,E2 24281.751} C_VEL
LIN {X 0,Y 536.468,Z 364.223,A -85,B 0,C 180,E1 24278.426,E2 24278.426} C_VEL
LIN {X 0,Y 536.426,Z 364.225,A -85,B 0,C 180,E1 24275.086,E2 24275.086} C_VEL
LIN {X 0,Y 536.427,Z 364.223,A -85,B 0,C 180,E1 24271.605,E2 24271.605} C_VEL
LIN {X 0,Y 536.466,Z 364.226,A -85,B 0,C 180,E1 24268.292,E2 24268.292} C_VEL
LIN {X 0,Y 536.427,Z 364.221,A -85,B 0,C 180,E1 24265.35,E2 24265.35} C_VEL
LIN {X 0,Y 535.437,Z 364.354,A -85,B 0,C 180,E1 24264.528,E2 24264.528} C_VEL
LIN {X 0,Y 528.977,Z 365.156,A -85,B 0,C 180,E1 24262.156,E2 24262.156} C_VEL
LIN {X 0,Y 528.516,Z 365.21,A -85,B 0,C 180,E1 24261.614,E2 24261.614} C_VEL
LIN {X 0,Y 528.523,Z 365.214,A -85,B 0,C 180,E1 24258.184,E2 24258.184} C_VEL
LIN {X 0,Y 528.493,Z 365.213,A -85,B 0,C 180,E1 24254.808,E2 24254.808} C_VEL
LIN {X 0,Y 528.529,Z 365.209,A -85,B 0,C 180,E1 24251.456,E2 24251.456} C_VEL
LIN {X 0,Y 528.525,Z 365.212,A -85,B 0,C 180,E1 24247.919,E2 24247.919} C_VEL
LIN {X 0,Y 528.497,Z 365.211,A -85,B 0,C 180,E1 24244.576,E2 24244.576} C_VEL
LIN {X 0,Y 528.522,Z 365.196,A -85,B 0,C 180,E1 24241.217,E2 24241.217} C_VEL
LIN {X 0,Y 528.522,Z 365.214,A -85,B 0,C 180,E1 24237.703,E2 24237.703} C_VEL
LIN {X 0,Y 528.503,Z 365.209,A -85,B 0,C 180,E1 24234.233,E2 24234.233} C_VEL
LIN {X 0,Y 528.519,Z 365.198,A -85,B 0,C 180,E1 24230.83,E2 24230.83} C_VEL
LIN {X 0,Y 528.519,Z 365.196,A -85,B 0,C 180,E1 24227.388,E2 24227.388} C_VEL
LIN {X 0,Y 528.505,Z 365.179,A -85,B 0,C 180,E1 24224.011,E2 24224.011} C_VEL
LIN {X 0,Y 528.55,Z 365.42,A -85,B 0,C 180,E1 24222.284,E2 24222.284} C_VEL
LIN {X 0,Y 528.971,Z 367.035,A -85,B 0,C 180,E1 24222.08,E2 24222.08} C_VEL
LIN {X 0,Y 531.021,Z 370.072,A -85,B 0,C 180,E1 24221.805,E2 24221.805} C_VEL
LIN {X 0,Y 532.212,Z 371.586,A -85,B 0,C 180,E1 24221.654,E2 24221.654} C_VEL
LIN {X 0,Y 535.023,Z 375.569,A -85,B 0,C 180,E1 24221.292,E2 24221.292} C_VEL
LIN {X 0,Y 545.828,Z 391.715,A -85,B 0,C 180,E1 24219.947,E2 24219.947} C_VEL
LIN {X 0,Y 543.148,Z 603.695,A -85,B 0,C 180,E1 24216.594,E2 24216.594} C_VEL
LIN {X 0,Y 541.797,Z 710.991,A -85,B 0,C 180,E1 24214.907,E2 24214.907} C_VEL
LIN {X 0,Y 541.052,Z 734.45,A -85,B 0,C 180,E1 24214.346,E2 24214.346} C_VEL
LIN {X 0,Y 540.082,Z 757.957,A -85,B 0,C 180,E1 24213.566,E2 24213.566} C_VEL
LIN {X 0,Y 539.025,Z 779.318,A -85,B 0,C 180,E1 24212.655,E2 24212.655} C_VEL
LIN {X 0,Y 537.729,Z 801.68,A -85,B 0,C 180,E1 24211.489,E2 24211.489} C_VEL
LIN {X 0,Y 536.477,Z 821.977,A -85,B 0,C 180,E1 24210.211,E2 24210.211} C_VEL
LIN {X 0,Y 535.033,Z 843.677,A -85,B 0,C 180,E1 24208.605,E2 24208.605} C_VEL
LIN {X 0,Y 533.715,Z 863.497,A -85,B 0,C 180,E1 24206.883,E2 24206.883} C_VEL
LIN {X 0,Y 532.447,Z 882.299,A -85,B 0,C 180,E1 24204.988,E2 24204.988} C_VEL
LIN {X 0,Y 531.324,Z 899.611,A -85,B 0,C 180,E1 24202.971,E2 24202.971} C_VEL
LIN {X 0,Y 530.365,Z 915.989,A -85,B 0,C 180,E1 24200.776,E2 24200.776} C_VEL
LIN {X 0,Y 529.567,Z 930.938,A -85,B 0,C 180,E1 24198.453,E2 24198.453} C_VEL
LIN {X 0,Y 528.957,Z 943.848,A -85,B 0,C 180,E1 24196.107,E2 24196.107} C_VEL
LIN {X 0,Y 528.508,Z 955.482,A -85,B 0,C 180,E1 24193.625,E2 24193.625} C_VEL
LIN {X 0,Y 528.226,Z 965.125,A -85,B 0,C 180,E1 24191.162,E2 24191.162} C_VEL
LIN {X 0,Y 528.04,Z 972.98,A -85,B 0,C 180,E1 24188.679,E2 24188.679} C_VEL
LIN {X 0,Y 527.936,Z 978.889,A -85,B 0,C 180,E1 24186.325,E2 24186.325} C_VEL
LIN {X 0,Y 527.897,Z 983.531,A -85,B 0,C 180,E1 24183.81,E2 24183.81} C_VEL
LIN {X 0,Y 527.91,Z 986.475,A -85,B 0,C 180,E1 24181.366,E2 24181.366} C_VEL
LIN {X 0,Y 527.909,Z 987.834,A -85,B 0,C 180,E1 24178.863,E2 24178.863} C_VEL
LIN {X 0,Y 527.896,Z 987.694,A -85,B 0,C 180,E1 24176.421,E2 24176.421} C_VEL
LIN {X 0,Y 527.906,Z 985.91,A -85,B 0,C 180,E1 24173.974,E2 24173.974} C_VEL
LIN {X 0,Y 527.924,Z 982.75,A -85,B 0,C 180,E1 24171.593,E2 24171.593} C_VEL
LIN {X 0,Y 527.951,Z 978,A -85,B 0,C 180,E1 24169.201,E2 24169.201} C_VEL
LIN {X 0,Y 528.057,Z 971.787,A -85,B 0,C 180,E1 24166.802,E2 24166.802} C_VEL
LIN {X 0,Y 528.268,Z 963.476,A -85,B 0,C 180,E1 24164.3,E2 24164.3} C_VEL
LIN {X 0,Y 528.577,Z 953.823,A -85,B 0,C 180,E1 24161.893,E2 24161.893} C_VEL
LIN {X 0,Y 529.011,Z 942.513,A -85,B 0,C 180,E1 24159.542,E2 24159.542} C_VEL
LIN {X 0,Y 529.653,Z 929.176,A -85,B 0,C 180,E1 24157.163,E2 24157.163} C_VEL
LIN {X 0,Y 530.457,Z 914.515,A -85,B 0,C 180,E1 24154.92,E2 24154.92} C_VEL
LIN {X 0,Y 531.389,Z 898.612,A -85,B 0,C 180,E1 24152.813,E2 24152.813} C_VEL
LIN {X 0,Y 532.547,Z 880.693,A -85,B 0,C 180,E1 24150.747,E2 24150.747} C_VEL
LIN {X 0,Y 533.86,Z 861.428,A -85,B 0,C 180,E1 24148.834,E2 24148.834} C_VEL
LIN {X 0,Y 535.121,Z 842.369,A -85,B 0,C 180,E1 24147.201,E2 24147.201} C_VEL
LIN {X 0,Y 536.498,Z 821.663,A -85,B 0,C 180,E1 24145.678,E2 24145.678} C_VEL
LIN {X 0,Y 537.803,Z 800.502,A -85,B 0,C 180,E1 24144.356,E2 24144.356} C_VEL
LIN {X 0,Y 539.073,Z 778.402,A -85,B 0,C 180,E1 24143.213,E2 24143.213} C_VEL
LIN {X 0,Y 540.135,Z 756.439,A -85,B 0,C 180,E1 24142.286,E2 24142.286} C_VEL
LIN {X 0,Y 541.099,Z 733.442,A -85,B 0,C 180,E1 24141.536,E2 24141.536} C_VEL
LIN {X 0,Y 541.826,Z 709.868,A -85,B 0,C 180,E1 24140.981,E2 24140.981} C_VEL
LIN {X 0,Y 544.494,Z 494.612,A -85,B 0,C 180,E1 24137.604,E2 24137.604} C_VEL
LIN {X 0,Y 545.655,Z 391.357,A -85,B 0,C 180,E1 24135.94,E2 24135.94} C_VEL
LIN {X 0,Y 534.552,Z 375.051,A -85,B 0,C 180,E1 24134.557,E2 24134.557} C_VEL
LIN {X 0,Y 531.948,Z 370.995,A -85,B 0,C 180,E1 24134.213,E2 24134.213} C_VEL
LIN {X 0,Y 529.259,Z 367.682,A -85,B 0,C 180,E1 24133.868,E2 24133.868} C_VEL
LIN {X 0,Y 528.666,Z 366.014,A -85,B 0,C 180,E1 24133.731,E2 24133.731} C_VEL
LIN {X 0,Y 528.524,Z 365.218,A -85,B 0,C 180,E1 24133.456,E2 24133.456} C_VEL
LIN {X 0,Y 528.517,Z 365.202,A -85,B 0,C 180,E1 24130.024,E2 24130.024} C_VEL
LIN {X 0,Y 528.511,Z 365.214,A -85,B 0,C 180,E1 24126.627,E2 24126.627} C_VEL
LIN {X 0,Y 528.521,Z 365.211,A -85,B 0,C 180,E1 24123.145,E2 24123.145} C_VEL
LIN {X 0,Y 528.506,Z 365.214,A -85,B 0,C 180,E1 24119.675,E2 24119.675} C_VEL
LIN {X 0,Y 528.522,Z 365.216,A -85,B 0,C 180,E1 24116.204,E2 24116.204} C_VEL
LIN {X 0,Y 528.527,Z 365.209,A -85,B 0,C 180,E1 24112.719,E2 24112.719} C_VEL
LIN {X 0,Y 528.491,Z 365.214,A -85,B 0,C 180,E1 24109.315,E2 24109.315} C_VEL
LIN {X 0,Y 528.518,Z 365.217,A -85,B 0,C 180,E1 24105.875,E2 24105.875} C_VEL
LIN {X 0,Y 528.519,Z 365.212,A -85,B 0,C 180,E1 24102.456,E2 24102.456} C_VEL
LIN {X 0,Y 528.476,Z 365.216,A -85,B 0,C 180,E1 24099.049,E2 24099.049} C_VEL
LIN {X 0,Y 528.514,Z 365.212,A -85,B 0,C 180,E1 24095.762,E2 24095.762} C_VEL
LIN {X 0,Y 528.48,Z 365.216,A -85,B 0,C 180,E1 24092.508,E2 24092.508} C_VEL
LIN {X 0,Y 528.465,Z 365.219,A -85,B 0,C 180,E1 24089.154,E2 24089.154} C_VEL
LIN {X 0,Y 528.521,Z 365.211,A -85,B 0,C 180,E1 24085.816,E2 24085.816} C_VEL
LIN {X 0,Y 528.451,Z 365.22,A -85,B 0,C 180,E1 24082.466,E2 24082.466} C_VEL
LIN {X 0,Y 528.449,Z 365.22,A -85,B 0,C 180,E1 24078.964,E2 24078.964} C_VEL
LIN {X 0,Y 528.487,Z 365.493,A -85,B 0,C 180,E1 24076.37,E2 24076.37} C_VEL
LIN {X 0,Y 529.938,Z 368.906,A -85,B 0,C 180,E1 24075.877,E2 24075.877} C_VEL
LIN {X 0,Y 540.226,Z 390.491,A -85,B 0,C 180,E1 24073.094,E2 24073.094} C_VEL
LIN {X 0,Y 543.309,Z 395.798,A -85,B 0,C 180,E1 24072.686,E2 24072.686} C_VEL
LIN {X 0,Y 545.986,Z 409.913,A -85,B 0,C 180,E1 24072.182,E2 24072.182} C_VEL
LIN {X 0,Y 543.35,Z 616.906,A -85,B 0,C 180,E1 24068.901,E2 24068.901} C_VEL
LIN {X 0,Y 541.8,Z 740.42,A -85,B 0,C 180,E1 24066.961,E2 24066.961} C_VEL
LIN {X 0,Y 541.062,Z 763.557,A -85,B 0,C 180,E1 24066.411,E2 24066.411} C_VEL
LIN {X 0,Y 540.18,Z 785.268,A -85,B 0,C 180,E1 24065.713,E2 24065.713} C_VEL
LIN {X 0,Y 539.163,Z 806.354,A -85,B 0,C 180,E1 24064.834,E2 24064.834} C_VEL
LIN {X 0,Y 538.07,Z 826.214,A -85,B 0,C 180,E1 24063.837,E2 24063.837} C_VEL
LIN {X 0,Y 536.756,Z 847.215,A -85,B 0,C 180,E1 24062.573,E2 24062.573} C_VEL
LIN {X 0,Y 535.491,Z 867.383,A -85,B 0,C 180,E1 24061.147,E2 24061.147} C_VEL
LIN {X 0,Y 534.112,Z 887.251,A -85,B 0,C 180,E1 24059.496,E2 24059.496} C_VEL
LIN {X 0,Y 532.814,Z 906.771,A -85,B 0,C 180,E1 24057.616,E2 24057.616} C_VEL
LIN {X 0,Y 531.723,Z 923.643,A -85,B 0,C 180,E1 24055.748,E2 24055.748} C_VEL
LIN {X 0,Y 530.695,Z 939.978,A -85,B 0,C 180,E1 24053.662,E2 24053.662} C_VEL
LIN {X 0,Y 529.87,Z 954.912,A -85,B 0,C 180,E1 24051.476,E2 24051.476} C_VEL
LIN {X 0,Y 529.23,Z 967.716,A -85,B 0,C 180,E1 24049.309,E2 24049.309} C_VEL
LIN {X 0,Y 528.701,Z 980.048,A -85,B 0,C 180,E1 24046.879,E2 24046.879} C_VEL
LIN {X 0,Y 528.369,Z 989.981,A -85,B 0,C 180,E1 24044.579,E2 24044.579} C_VEL
LIN {X 0,Y 528.129,Z 998.692,A -85,B 0,C 180,E1 24042.133,E2 24042.133} C_VEL
LIN {X 0,Y 527.98,Z 1005.767,A -85,B 0,C 180,E1 24039.706,E2 24039.706} C_VEL
LIN {X 0,Y 527.919,Z 1010.836,A -85,B 0,C 180,E1 24037.402,E2 24037.402} C_VEL
LIN {X 0,Y 527.917,Z 1014.432,A -85,B 0,C 180,E1 24035.219,E2 24035.219} C_VEL
LIN {X 0,Y 527.909,Z 1017.054,A -85,B 0,C 180,E1 24032.608,E2 24032.608} C_VEL
LIN {X 0,Y 527.891,Z 1017.939,A -85,B 0,C 180,E1 24030.328,E2 24030.328} C_VEL
LIN {X 0,Y 527.914,Z 1017.326,A -85,B 0,C 180,E1 24027.832,E2 24027.832} C_VEL
LIN {X 0,Y 527.905,Z 1015.392,A -85,B 0,C 180,E1 24025.549,E2 24025.549} C_VEL
LIN {X 0,Y 527.909,Z 1011.673,A -85,B 0,C 180,E1 24023.041,E2 24023.041} C_VEL
LIN {X 0,Y 527.986,Z 1007.07,A -85,B 0,C 180,E1 24020.85,E2 24020.85} C_VEL
LIN {X 0,Y 528.099,Z 1000.128,A -85,B 0,C 180,E1 24018.315,E2 24018.315} C_VEL
LIN {X 0,Y 528.269,Z 992.535,A -85,B 0,C 180,E1 24016.095,E2 24016.095} C_VEL
LIN {X 0,Y 528.602,Z 982.413,A -85,B 0,C 180,E1 24013.634,E2 24013.634} C_VEL
LIN {X 0,Y 529.042,Z 971.426,A -85,B 0,C 180,E1 24011.377,E2 24011.377} C_VEL
LIN {X 0,Y 529.661,Z 958.484,A -85,B 0,C 180,E1 24009.101,E2 24009.101} C_VEL
LIN {X 0,Y 530.477,Z 944.055,A -85,B 0,C 180,E1 24006.895,E2 24006.895} C_VEL
LIN {X 0,Y 531.404,Z 928.335,A -85,B 0,C 180,E1 24004.825,E2 24004.825} C_VEL
LIN {X 0,Y 532.569,Z 910.157,A -85,B 0,C 180,E1 24002.74,E2 24002.74} C_VEL
LIN {X 0,Y 533.836,Z 891.948,A -85,B 0,C 180,E1 24000.924,E2 24000.924} C_VEL
LIN {X 0,Y 535.097,Z 872.564,A -85,B 0,C 180,E1 23999.264,E2 23999.264} C_VEL
LIN {X 0,Y 536.493,Z 851.793,A -85,B 0,C 180,E1 23997.732,E2 23997.732} C_VEL
LIN {X 0,Y 537.704,Z 831.889,A -85,B 0,C 180,E1 23996.482,E2 23996.482} C_VEL
LIN {X 0,Y 538.956,Z 810.342,A -85,B 0,C 180,E1 23995.351,E2 23995.351} C_VEL
LIN {X 0,Y 539.928,Z 791.09,A -85,B 0,C 180,E1 23994.516,E2 23994.516} C_VEL
LIN {X 0,Y 540.899,Z 767.522,A -85,B 0,C 180,E1 23993.702,E2 23993.702} C_VEL
LIN {X 0,Y 541.637,Z 746.118,A -85,B 0,C 180,E1 23993.155,E2 23993.155} C_VEL
LIN {X 0,Y 542.201,Z 714.347,A -85,B 0,C 180,E1 23992.61,E2 23992.61} C_VEL
LIN {X 0,Y 544.76,Z 503.698,A -85,B 0,C 180,E1 23989.318,E2 23989.318} C_VEL
LIN {X 0,Y 545.826,Z 408.075,A -85,B 0,C 180,E1 23987.771,E2 23987.771} C_VEL
LIN {X 0,Y 542.89,Z 394.737,A -85,B 0,C 180,E1 23987.255,E2 23987.255} C_VEL
LIN {X 0,Y 540.028,Z 390.004,A -85,B 0,C 180,E1 23986.843,E2 23986.843} C_VEL
LIN {X 0,Y 530.102,Z 369.086,A -85,B 0,C 180,E1 23984.106,E2 23984.106} C_VEL
LIN {X 0,Y 528.493,Z 365.477,A -85,B 0,C 180,E1 23983.571,E2 23983.571} C_VEL
LIN {X 0,Y 528.477,Z 365.212,A -85,B 0,C 180,E1 23981.902,E2 23981.902} C_VEL
LIN {X 0,Y 528.463,Z 365.201,A -85,B 0,C 180,E1 23978.774,E2 23978.774} C_VEL
LIN {X 0,Y 528.446,Z 365.196,A -85,B 0,C 180,E1 23975.373,E2 23975.373} C_VEL
LIN {X 0,Y 528.515,Z 365.211,A -85,B 0,C 180,E1 23972.064,E2 23972.064} C_VEL
LIN {X 0,Y 528.438,Z 365.213,A -85,B 0,C 180,E1 23968.841,E2 23968.841} C_VEL
LIN {X 0,Y 528.478,Z 365.218,A -85,B 0,C 180,E1 23965.527,E2 23965.527} C_VEL
LIN {X 0,Y 528.459,Z 365.215,A -85,B 0,C 180,E1 23962.314,E2 23962.314} C_VEL
LIN {X 0,Y 528.449,Z 365.219,A -85,B 0,C 180,E1 23958.877,E2 23958.877} C_VEL
LIN {X 0,Y 528.52,Z 365.216,A -85,B 0,C 180,E1 23955.583,E2 23955.583} C_VEL
LIN {X 0,Y 528.452,Z 365.218,A -85,B 0,C 180,E1 23952.345,E2 23952.345} C_VEL
LIN {X 0,Y 528.479,Z 365.214,A -85,B 0,C 180,E1 23948.925,E2 23948.925} C_VEL
LIN {X 0,Y 528.481,Z 365.218,A -85,B 0,C 180,E1 23945.755,E2 23945.755} C_VEL
LIN {X 0,Y 528.462,Z 365.215,A -85,B 0,C 180,E1 23942.385,E2 23942.385} C_VEL
LIN {X 0,Y 528.527,Z 365.213,A -85,B 0,C 180,E1 23939.132,E2 23939.132} C_VEL
LIN {X 0,Y 528.468,Z 365.217,A -85,B 0,C 180,E1 23935.768,E2 23935.768} C_VEL
LIN {X 0,Y 528.477,Z 365.214,A -85,B 0,C 180,E1 23932.28,E2 23932.28} C_VEL
LIN {X 0,Y 528.519,Z 365.217,A -85,B 0,C 180,E1 23928.984,E2 23928.984} C_VEL
LIN {X 0,Y 528.472,Z 365.215,A -85,B 0,C 180,E1 23925.606,E2 23925.606} C_VEL
LIN {X 0,Y 528.509,Z 365.212,A -85,B 0,C 180,E1 23922.266,E2 23922.266} C_VEL
LIN {X 0,Y 528.504,Z 365.212,A -85,B 0,C 180,E1 23918.933,E2 23918.933} C_VEL
LIN {X 0,Y 528.478,Z 365.212,A -85,B 0,C 180,E1 23915.522,E2 23915.522} C_VEL
LIN {X 0,Y 528.527,Z 365.211,A -85,B 0,C 180,E1 23912.142,E2 23912.142} C_VEL
LIN {X 0,Y 528.501,Z 365.211,A -85,B 0,C 180,E1 23908.765,E2 23908.765} C_VEL
LIN {X 0,Y 528.486,Z 365.21,A -85,B 0,C 180,E1 23905.286,E2 23905.286} C_VEL
LIN {X 0,Y 528.528,Z 365.211,A -85,B 0,C 180,E1 23901.897,E2 23901.897} C_VEL
LIN {X 0,Y 528.516,Z 365.21,A -85,B 0,C 180,E1 23901.614,E2 23901.614} C_VEL
LIN {X 0,Y 527.493,Z 365.34,A -85,B 0,C 180,E1 23900.78,E2 23900.78} C_VEL
LIN {X 0,Y 521.113,Z 366.14,A -85,B 0,C 180,E1 23898.434,E2 23898.434} C_VEL
LIN {X 0,Y 520.585,Z 366.201,A -85,B 0,C 180,E1 23897.823,E2 23897.823} C_VEL
LIN {X 0,Y 520.571,Z 366.205,A -85,B 0,C 180,E1 23894.351,E2 23894.351} C_VEL
LIN {X 0,Y 520.556,Z 366.202,A -85,B 0,C 180,E1 23890.819,E2 23890.819} C_VEL
LIN {X 0,Y 520.582,Z 366.196,A -85,B 0,C 180,E1 23887.501,E2 23887.501} C_VEL
LIN {X 0,Y 520.58,Z 366.2,A -85,B 0,C 180,E1 23883.976,E2 23883.976} C_VEL
LIN {X 0,Y 520.559,Z 366.183,A -85,B 0,C 180,E1 23880.465,E2 23880.465} C_VEL
LIN {X 0,Y 520.583,Z 366.194,A -85,B 0,C 180,E1 23877.073,E2 23877.073} C_VEL
LIN {X 0,Y 520.586,Z 366.205,A -85,B 0,C 180,E1 23873.542,E2 23873.542} C_VEL
LIN {X 0,Y 520.566,Z 366.196,A -85,B 0,C 180,E1 23870.077,E2 23870.077} C_VEL
LIN {X 0,Y 520.584,Z 366.187,A -85,B 0,C 180,E1 23866.583,E2 23866.583} C_VEL
LIN {X 0,Y 520.594,Z 366.305,A -85,B 0,C 180,E1 23863.156,E2 23863.156} C_VEL
LIN {X 0,Y 520.936,Z 367.746,A -85,B 0,C 180,E1 23862.939,E2 23862.939} C_VEL
LIN {X 0,Y 522.889,Z 370.856,A -85,B 0,C 180,E1 23862.658,E2 23862.658} C_VEL
LIN {X 0,Y 524.255,Z 372.416,A -85,B 0,C 180,E1 23862.48,E2 23862.48} C_VEL
LIN {X 0,Y 527.026,Z 376.445,A -85,B 0,C 180,E1 23862.106,E2 23862.106} C_VEL
LIN {X 0,Y 539.834,Z 395.169,A -85,B 0,C 180,E1 23860.461,E2 23860.461} C_VEL
LIN {X 0,Y 536.824,Z 609.564,A -85,B 0,C 180,E1 23857.036,E2 23857.036} C_VEL
LIN {X 0,Y 535.396,Z 711.054,A -85,B 0,C 180,E1 23855.422,E2 23855.422} C_VEL
LIN {X 0,Y 534.602,Z 734.211,A -85,B 0,C 180,E1 23854.865,E2 23854.865} C_VEL
LIN {X 0,Y 533.518,Z 757.591,A -85,B 0,C 180,E1 23854.088,E2 23854.088} C_VEL
LIN {X 0,Y 532.372,Z 778.929,A -85,B 0,C 180,E1 23853.173,E2 23853.173} C_VEL
LIN {X 0,Y 531.004,Z 800.429,A -85,B 0,C 180,E1 23852.047,E2 23852.047} C_VEL
LIN {X 0,Y 529.586,Z 820.992,A -85,B 0,C 180,E1 23850.754,E2 23850.754} C_VEL
LIN {X 0,Y 528.048,Z 842.175,A -85,B 0,C 180,E1 23849.183,E2 23849.183} C_VEL
LIN {X 0,Y 526.548,Z 862.23,A -85,B 0,C 180,E1 23847.44,E2 23847.44} C_VEL
LIN {X 0,Y 525.105,Z 881.22,A -85,B 0,C 180,E1 23845.52,E2 23845.52} C_VEL
LIN {X 0,Y 523.822,Z 899.106,A -85,B 0,C 180,E1 23843.421,E2 23843.421} C_VEL
LIN {X 0,Y 522.776,Z 914.785,A -85,B 0,C 180,E1 23841.307,E2 23841.307} C_VEL
LIN {X 0,Y 521.88,Z 929.225,A -85,B 0,C 180,E1 23839.064,E2 23839.064} C_VEL
LIN {X 0,Y 521.167,Z 942.354,A -85,B 0,C 180,E1 23836.688,E2 23836.688} C_VEL
LIN {X 0,Y 520.673,Z 953.734,A -85,B 0,C 180,E1 23834.288,E2 23834.288} C_VEL
LIN {X 0,Y 520.313,Z 963.765,A -85,B 0,C 180,E1 23831.744,E2 23831.744} C_VEL
LIN {X 0,Y 520.075,Z 972.118,A -85,B 0,C 180,E1 23829.163,E2 23829.163} C_VEL
LIN {X 0,Y 519.962,Z 978.142,A -85,B 0,C 180,E1 23826.781,E2 23826.781} C_VEL
LIN {X 0,Y 519.917,Z 983.029,A -85,B 0,C 180,E1 23824.236,E2 23824.236} C_VEL
LIN {X 0,Y 519.913,Z 986.176,A -85,B 0,C 180,E1 23821.739,E2 23821.739} C_VEL
LIN {X 0,Y 519.917,Z 987.789,A -85,B 0,C 180,E1 23819.103,E2 23819.103} C_VEL
LIN {X 0,Y 519.91,Z 987.781,A -85,B 0,C 180,E1 23816.762,E2 23816.762} C_VEL
LIN {X 0,Y 519.912,Z 986.228,A -85,B 0,C 180,E1 23814.221,E2 23814.221} C_VEL
LIN {X 0,Y 519.918,Z 983.049,A -85,B 0,C 180,E1 23811.687,E2 23811.687} C_VEL
LIN {X 0,Y 519.959,Z 978.236,A -85,B 0,C 180,E1 23809.169,E2 23809.169} C_VEL
LIN {X 0,Y 520.072,Z 972.193,A -85,B 0,C 180,E1 23806.773,E2 23806.773} C_VEL
LIN {X 0,Y 520.308,Z 963.918,A -85,B 0,C 180,E1 23804.209,E2 23804.209} C_VEL
LIN {X 0,Y 520.643,Z 954.441,A -85,B 0,C 180,E1 23801.789,E2 23801.789} C_VEL
LIN {X 0,Y 521.137,Z 943.03,A -85,B 0,C 180,E1 23799.356,E2 23799.356} C_VEL
LIN {X 0,Y 521.846,Z 929.934,A -85,B 0,C 180,E1 23796.966,E2 23796.966} C_VEL
LIN {X 0,Y 522.75,Z 915.219,A -85,B 0,C 180,E1 23794.667,E2 23794.667} C_VEL
LIN {X 0,Y 523.772,Z 899.753,A -85,B 0,C 180,E1 23792.57,E2 23792.57} C_VEL
LIN {X 0,Y 525.033,Z 882.215,A -85,B 0,C 180,E1 23790.499,E2 23790.499} C_VEL
LIN {X 0,Y 526.451,Z 863.553,A -85,B 0,C 180,E1 23788.595,E2 23788.595} C_VEL
LIN {X 0,Y 527.911,Z 843.874,A -85,B 0,C 180,E1 23786.863,E2 23786.863} C_VEL
LIN {X 0,Y 529.484,Z 822.56,A -85,B 0,C 180,E1 23785.263,E2 23785.263} C_VEL
LIN {X 0,Y 530.905,Z 801.971,A -85,B 0,C 180,E1 23783.951,E2 23783.951} C_VEL
LIN {X 0,Y 532.303,Z 780.122,A -85,B 0,C 180,E1 23782.794,E2 23782.794} C_VEL
LIN {X 0,Y 533.488,Z 758.285,A -85,B 0,C 180,E1 23781.849,E2 23781.849} C_VEL
LIN {X 0,Y 534.582,Z 734.69,A -85,B 0,C 180,E1 23781.059,E2 23781.059} C_VEL
LIN {X 0,Y 535.383,Z 711.538,A -85,B 0,C 180,E1 23780.498,E2 23780.498} C_VEL
LIN {X 0,Y 536.451,Z 637.527,A -85,B 0,C 180,E1 23779.312,E2 23779.312} C_VEL
LIN {X 0,Y 539.362,Z 427.294,A -85,B 0,C 180,E1 23775.969,E2 23775.969} C_VEL
LIN {X 0,Y 539.699,Z 394.954,A -85,B 0,C 180,E1 23775.432,E2 23775.432} C_VEL
LIN {X 0,Y 529.67,Z 380.365,A -85,B 0,C 180,E1 23774.15,E2 23774.15} C_VEL
LIN {X 0,Y 526.523,Z 375.878,A -85,B 0,C 180,E1 23773.732,E2 23773.732} C_VEL
LIN {X 0,Y 523.597,Z 371.491,A -85,B 0,C 180,E1 23773.332,E2 23773.332} C_VEL
LIN {X 0,Y 521.3,Z 368.675,A -85,B 0,C 180,E1 23773.025,E2 23773.025} C_VEL
LIN {X 0,Y 520.693,Z 366.938,A -85,B 0,C 180,E1 23772.871,E2 23772.871} C_VEL
LIN {X 0,Y 520.573,Z 366.24,A -85,B 0,C 180,E1 23772.648,E2 23772.648} C_VEL
LIN {X 0,Y 520.58,Z 366.203,A -85,B 0,C 180,E1 23769.164,E2 23769.164} C_VEL
LIN {X 0,Y 520.573,Z 366.205,A -85,B 0,C 180,E1 23765.732,E2 23765.732} C_VEL
LIN {X 0,Y 520.583,Z 366.2,A -85,B 0,C 180,E1 23762.202,E2 23762.202} C_VEL
LIN {X 0,Y 520.581,Z 366.202,A -85,B 0,C 180,E1 23758.68,E2 23758.68} C_VEL
LIN {X 0,Y 520.562,Z 366.196,A -85,B 0,C 180,E1 23755.263,E2 23755.263} C_VEL
LIN {X 0,Y 520.565,Z 366.206,A -85,B 0,C 180,E1 23751.718,E2 23751.718} C_VEL
LIN {X 0,Y 520.586,Z 366.203,A -85,B 0,C 180,E1 23748.254,E2 23748.254} C_VEL
LIN {X 0,Y 520.556,Z 366.201,A -85,B 0,C 180,E1 23744.858,E2 23744.858} C_VEL
LIN {X 0,Y 520.547,Z 366.205,A -85,B 0,C 180,E1 23741.407,E2 23741.407} C_VEL
LIN {X 0,Y 520.592,Z 366.203,A -85,B 0,C 180,E1 23738.006,E2 23738.006} C_VEL
LIN {X 0,Y 520.54,Z 366.205,A -85,B 0,C 180,E1 23734.638,E2 23734.638} C_VEL
LIN {X 0,Y 520.528,Z 366.203,A -85,B 0,C 180,E1 23731.155,E2 23731.155} C_VEL
LIN {X 0,Y 520.582,Z 366.199,A -85,B 0,C 180,E1 23727.858,E2 23727.858} C_VEL
LIN {X 0,Y 520.516,Z 366.209,A -85,B 0,C 180,E1 23724.536,E2 23724.536} C_VEL
LIN {X 0,Y 520.516,Z 366.207,A -85,B 0,C 180,E1 23721.076,E2 23721.076} C_VEL
LIN {X 0,Y 520.549,Z 366.204,A -85,B 0,C 180,E1 23717.854,E2 23717.854} C_VEL
LIN {X 0,Y 520.594,Z 366.642,A -85,B 0,C 180,E1 23717.12,E2 23717.12} C_VEL
LIN {X 0,Y 522.255,Z 370.328,A -85,B 0,C 180,E1 23716.583,E2 23716.583} C_VEL
LIN {X 0,Y 532.058,Z 390.698,A -85,B 0,C 180,E1 23713.897,E2 23713.897} C_VEL
LIN {X 0,Y 537.867,Z 400.139,A -85,B 0,C 180,E1 23713.135,E2 23713.135} C_VEL
LIN {X 0,Y 540.01,Z 411.676,A -85,B 0,C 180,E1 23712.723,E2 23712.723} C_VEL
LIN {X 0,Y 537.105,Z 618.464,A -85,B 0,C 180,E1 23709.414,E2 23709.414} C_VEL
LIN {X 0,Y 535.404,Z 740.425,A -85,B 0,C 180,E1 23707.477,E2 23707.477} C_VEL
LIN {X 0,Y 534.606,Z 763.425,A -85,B 0,C 180,E1 23706.927,E2 23706.927} C_VEL
LIN {X 0,Y 533.654,Z 784.625,A -85,B 0,C 180,E1 23706.243,E2 23706.243} C_VEL
LIN {X 0,Y 532.492,Z 806.35,A -85,B 0,C 180,E1 23705.335,E2 23705.335} C_VEL
LIN {X 0,Y 531.277,Z 826.54,A -85,B 0,C 180,E1 23704.311,E2 23704.311} C_VEL
LIN {X 0,Y 529.773,Z 848.112,A -85,B 0,C 180,E1 23702.992,E2 23702.992} C_VEL
LIN {X 0,Y 528.375,Z 868.162,A -85,B 0,C 180,E1 23701.551,E2 23701.551} C_VEL
LIN {X 0,Y 526.897,Z 887.249,A -85,B 0,C 180,E1 23699.941,E2 23699.941} C_VEL
LIN {X 0,Y 525.421,Z 907.14,A -85,B 0,C 180,E1 23697.997,E2 23697.997} C_VEL
LIN {X 0,Y 524.214,Z 923.642,A -85,B 0,C 180,E1 23696.144,E2 23696.144} C_VEL
LIN {X 0,Y 523.075,Z 939.976,A -85,B 0,C 180,E1 23694.028,E2 23694.028} C_VEL
LIN {X 0,Y 522.123,Z 955.233,A -85,B 0,C 180,E1 23691.758,E2 23691.758} C_VEL
LIN {X 0,Y 521.411,Z 967.714,A -85,B 0,C 180,E1 23689.61,E2 23689.61} C_VEL
LIN {X 0,Y 520.804,Z 980.315,A -85,B 0,C 180,E1 23687.084,E2 23687.084} C_VEL
LIN {X 0,Y 520.424,Z 990.439,A -85,B 0,C 180,E1 23684.693,E2 23684.693} C_VEL
LIN {X 0,Y 520.153,Z 999.049,A -85,B 0,C 180,E1 23682.21,E2 23682.21} C_VEL
LIN {X 0,Y 519.988,Z 1006.036,A -85,B 0,C 180,E1 23679.745,E2 23679.745} C_VEL
LIN {X 0,Y 519.921,Z 1011.043,A -85,B 0,C 180,E1 23677.406,E2 23677.406} C_VEL
LIN {X 0,Y 519.915,Z 1014.751,A -85,B 0,C 180,E1 23675.078,E2 23675.078} C_VEL
LIN {X 0,Y 519.911,Z 1017.121,A -85,B 0,C 180,E1 23672.538,E2 23672.538} C_VEL
LIN {X 0,Y 519.905,Z 1017.983,A -85,B 0,C 180,E1 23670.113,E2 23670.113} C_VEL
LIN {X 0,Y 519.914,Z 1017.259,A -85,B 0,C 180,E1 23667.688,E2 23667.688} C_VEL
LIN {X 0,Y 519.905,Z 1015.165,A -85,B 0,C 180,E1 23665.26,E2 23665.26} C_VEL
LIN {X 0,Y 519.912,Z 1011.467,A -85,B 0,C 180,E1 23662.822,E2 23662.822} C_VEL
LIN {X 0,Y 519.989,Z 1007.07,A -85,B 0,C 180,E1 23660.708,E2 23660.708} C_VEL
LIN {X 0,Y 520.134,Z 999.968,A -85,B 0,C 180,E1 23658.083,E2 23658.083} C_VEL
LIN {X 0,Y 520.349,Z 992.127,A -85,B 0,C 180,E1 23655.765,E2 23655.765} C_VEL
